C05489=1201.609,-125.840,-37.789,179.030,5.510,149.258
C05490=1201.614,-126.089,-37.779,179.027,5.510,149.259
C05491=1201.619,-126.339,-37.770,179.026,5.510,149.259
C05492=1201.624,-126.589,-37.761,179.024,5.510,149.260
C05493=1201.631,-126.838,-37.752,179.022,5.509,149.261
C05494=1201.208,-126.849,-37.790,179.017,5.513,149.263
C05495=1201.203,-126.600,-37.800,179.020,5.513,149.262
C05496=1201.198,-126.350,-37.809,179.021,5.513,149.262
C05497=1201.192,-126.100,-37.818,179.024,5.514,149.261
C05498=1201.187,-125.850,-37.827,179.026,5.513,149.260
C05499=1201.182,-125.601,-37.836,179.028,5.513,149.260
C05500=1201.176,-125.350,-37.845,179.030,5.514,149.259
C05501=1201.171,-125.101,-37.855,179.032,5.514,149.258
C05502=1201.166,-124.851,-37.864,179.035,5.514,149.258
C05503=1201.161,-124.601,-37.873,179.037,5.514,149.257
C05504=1201.155,-124.351,-37.882,179.039,5.515,149.257
C05505=1201.150,-124.101,-37.891,179.041,5.514,149.256
C05506=1201.145,-123.852,-37.901,179.044,5.515,149.255
C05507=1201.140,-123.602,-37.910,179.045,5.515,149.255
C05508=1201.134,-123.352,-37.919,179.048,5.515,149.254
C05509=1201.129,-123.102,-37.928,179.050,5.515,149.253
C05510=1201.124,-122.853,-37.938,179.052,5.515,149.253
C05511=1201.118,-122.603,-37.947,179.054,5.515,149.252
C05512=1201.113,-122.353,-37.956,179.057,5.516,149.251
C05513=1201.108,-122.103,-37.965,179.059,5.515,149.251
C05514=1201.103,-121.854,-37.974,179.060,5.515,149.250
C05515=1201.097,-121.604,-37.984,179.063,5.516,149.250
C05516=1201.092,-121.354,-37.993,179.065,5.515,149.249
C05517=1201.087,-121.105,-38.002,179.067,5.516,149.248
C05518=1201.081,-120.855,-38.012,179.069,5.516,149.248
C05519=1201.076,-120.605,-38.021,179.072,5.516,149.247
C05520=1201.071,-120.355,-38.030,179.074,5.516,149.246
C05521=1201.065,-120.105,-38.040,179.076,5.516,149.246
C05522=1201.060,-119.855,-38.049,179.078,5.516,149.245
C05523=1201.055,-119.606,-38.058,179.081,5.517,149.245
C05524=1201.049,-119.356,-38.068,179.083,5.516,149.244
C05525=1201.044,-119.106,-38.077,179.085,5.517,149.243
C05526=1201.039,-118.857,-38.086,179.087,5.517,149.243
C05527=1201.033,-118.607,-38.096,179.090,5.517,149.242
C05528=1201.028,-118.357,-38.105,179.091,5.517,149.241
C05529=1201.023,-118.108,-38.114,179.094,5.518,149.241
C05530=1201.017,-117.858,-38.124,179.096,5.517,149.240
C05531=1201.012,-117.608,-38.134,179.098,5.518,149.239
C05532=1201.007,-117.358,-38.143,179.100,5.518,149.239
C05533=1201.001,-117.108,-38.152,179.102,5.518,149.238
C05534=1200.997,-116.859,-38.162,179.105,5.518,149.238
C05535=1200.991,-116.608,-38.171,179.107,5.518,149.237
C05536=1200.986,-116.359,-38.181,179.109,5.518,149.236
C05537=1200.980,-116.109,-38.191,179.111,5.518,149.236
C05538=1200.975,-115.859,-38.199,179.114,5.518,149.235
C05539=1200.970,-115.610,-38.209,179.115,5.518,149.234
C05540=1200.965,-115.360,-38.219,179.118,5.519,149.234
C05541=1200.960,-115.110,-38.228,179.120,5.518,149.233
C05542=1200.954,-114.860,-38.238,179.122,5.519,149.233
C05543=1200.949,-114.611,-38.247,179.124,5.519,149.232
C05544=1200.943,-114.361,-38.257,179.127,5.519,149.231
C05545=1200.938,-114.112,-38.266,179.128,5.519,149.231
C05546=1200.932,-113.861,-38.276,179.131,5.520,149.230
C05547=1200.928,-113.611,-38.286,179.133,5.519,149.229
C05548=1200.923,-113.362,-38.295,179.135,5.520,149.229
C05549=1200.917,-113.112,-38.305,179.138,5.520,149.228
C05550=1200.912,-112.862,-38.314,179.140,5.520,149.227
C05551=1200.906,-112.613,-38.324,179.142,5.520,149.227
C05552=1200.901,-112.363,-38.333,179.145,5.520,149.226
C05553=1200.896,-112.113,-38.343,179.147,5.520,149.225
C05554=1200.890,-111.863,-38.352,179.149,5.521,149.225
C05555=1200.885,-111.614,-38.362,179.151,5.520,149.224
C05556=1200.880,-111.363,-38.372,179.153,5.521,149.224
C05557=1200.875,-111.114,-38.382,179.155,5.521,149.223
C05558=1200.870,-110.865,-38.391,179.158,5.521,149.222
C05559=1200.864,-110.614,-38.401,179.160,5.521,149.222
C05560=1200.859,-110.365,-38.410,179.162,5.522,149.221
C05561=1200.853,-110.115,-38.420,179.164,5.521,149.220
C05562=1200.848,-109.866,-38.430,179.167,5.522,149.220
C05563=1200.843,-109.615,-38.439,179.168,5.522,149.219
C05564=1200.838,-109.366,-38.449,179.171,5.522,149.218
C05565=1200.833,-109.116,-38.459,179.173,5.522,149.218
C05566=1200.827,-108.866,-38.469,179.175,5.522,149.217
C05567=1200.822,-108.617,-38.478,179.178,5.522,149.217
C05568=1200.816,-108.367,-38.489,179.180,5.522,149.216
C05569=1200.812,-108.117,-38.498,179.182,5.522,149.215
C05570=1200.806,-107.867,-38.508,179.184,5.523,149.215
C05571=1200.801,-107.618,-38.518,179.187,5.522,149.214
C05572=1200.795,-107.368,-38.527,179.189,5.523,149.213
C05573=1200.790,-107.118,-38.537,179.191,5.523,149.213
C05574=1200.785,-106.868,-38.547,179.194,5.523,149.212
C05575=1200.780,-106.618,-38.557,179.195,5.523,149.211
C05576=1200.775,-106.369,-38.566,179.198,5.524,149.211
C05577=1200.769,-106.119,-38.577,179.200,5.523,149.210
C05578=1200.764,-105.869,-38.586,179.202,5.524,149.210
C05579=1200.759,-105.619,-38.596,179.204,5.524,149.209
C05580=1200.753,-105.370,-38.606,179.207,5.524,149.208
C05581=1200.748,-105.120,-38.615,179.208,5.524,149.208
C05582=1200.743,-104.870,-38.625,179.211,5.524,149.207
C05583=1200.737,-104.621,-38.636,179.213,5.524,149.206
C05584=1200.733,-104.371,-38.646,179.216,5.525,149.206
C05585=1200.727,-104.121,-38.655,179.217,5.525,149.205
C05586=1200.722,-103.871,-38.665,179.220,5.525,149.204
C05587=1200.716,-103.622,-38.675,179.222,5.525,149.204
C05588=1200.711,-103.372,-38.685,179.224,5.525,149.203
C05589=1200.706,-103.122,-38.694,179.226,5.525,149.202
C05590=1200.701,-102.872,-38.705,179.229,5.525,149.202
C05591=1200.695,-102.623,-38.715,179.231,5.525,149.201
C05592=1200.691,-102.373,-38.725,179.233,5.526,149.200
C05593=1200.685,-102.123,-38.735,179.236,5.525,149.200
C05594=1200.679,-101.873,-38.744,179.238,5.526,149.199
C05595=1200.674,-101.602,-38.755,179.240,5.527,149.199
C05596=1200.669,-101.330,-38.766,179.242,5.526,149.198
C05597=1200.662,-101.060,-38.778,179.245,5.527,149.197
C05598=1200.657,-100.788,-38.788,179.248,5.527,149.196
C05599=1200.651,-100.538,-38.798,179.250,5.527,149.196
C05600=1200.646,-100.288,-38.809,179.253,5.527,149.195
C05601=1200.641,-100.039,-38.818,179.254,5.527,149.195
C05602=1200.636,-99.789,-38.828,179.257,5.527,149.194
C05603=1200.631,-99.539,-38.839,179.259,5.527,149.193
C05604=1200.626,-99.289,-38.848,179.262,5.527,149.192
C05605=1200.620,-99.039,-38.858,179.263,5.527,149.192
C05606=1200.614,-98.790,-38.868,179.266,5.528,149.191
C05607=1200.609,-98.540,-38.879,179.268,5.527,149.190
C05608=1200.605,-98.290,-38.888,179.270,5.528,149.190
C05609=1200.599,-98.041,-38.899,179.272,5.528,149.189
C05610=1200.594,-97.791,-38.909,179.275,5.528,149.189
C05611=1200.588,-97.541,-38.919,179.277,5.528,149.188
C05612=1200.583,-97.292,-38.930,179.279,5.529,149.187
C05613=1200.578,-97.042,-38.940,179.282,5.529,149.187
C05614=1200.573,-96.792,-38.950,179.284,5.529,149.186
C05615=1200.567,-96.542,-38.959,179.286,5.530,149.185
C05616=1200.562,-96.292,-38.970,179.288,5.529,149.185
C05617=1200.556,-96.042,-38.980,179.291,5.530,149.184
C05618=1200.552,-95.793,-38.990,179.293,5.529,149.183
C05619=1200.547,-95.543,-39.000,179.295,5.530,149.183
C05620=1200.541,-95.293,-39.011,179.297,5.530,149.182
C05621=1200.535,-95.044,-39.021,179.300,5.530,149.181
C05622=1200.530,-94.793,-39.031,179.302,5.530,149.181
C05623=1200.525,-94.544,-39.041,179.304,5.530,149.180
C05624=1200.520,-94.295,-39.051,179.306,5.530,149.180
C05625=1200.515,-94.044,-39.062,179.309,5.530,149.179
C05626=1200.509,-93.795,-39.072,179.311,5.530,149.178
C05627=1200.504,-93.545,-39.082,179.313,5.531,149.178
C05628=1200.499,-93.295,-39.093,179.316,5.531,149.177
C05629=1200.494,-93.046,-39.102,179.318,5.531,149.176
C05630=1200.489,-92.796,-39.114,179.320,5.532,149.176
C05631=1200.484,-92.547,-39.124,179.322,5.531,149.175
C05632=1200.478,-92.297,-39.134,179.325,5.532,149.174
C05633=1200.473,-92.047,-39.145,179.327,5.532,149.174
C05634=1200.467,-91.797,-39.155,179.329,5.532,149.173
C05635=1200.462,-91.548,-39.165,179.331,5.532,149.172
C05636=1200.457,-91.297,-39.176,179.334,5.532,149.172
C05637=1200.452,-91.048,-39.185,179.336,5.532,149.171
C05638=1200.447,-90.798,-39.196,179.338,5.533,149.170
C05639=1200.441,-90.548,-39.206,179.341,5.533,149.170
C05640=1200.436,-90.299,-39.216,179.343,5.533,149.169
C05641=1200.431,-90.049,-39.227,179.345,5.533,149.169
C05642=1200.425,-89.800,-39.238,179.347,5.533,149.168
C05643=1200.420,-89.549,-39.248,179.350,5.534,149.167
C05644=1200.415,-89.300,-39.258,179.352,5.533,149.166
C05645=1200.410,-89.050,-39.269,179.354,5.534,149.166
C05646=1200.404,-88.800,-39.279,179.356,5.534,149.165
C05647=1200.399,-88.551,-39.289,179.359,5.534,149.165
C05648=1200.394,-88.301,-39.301,179.361,5.534,149.164
C05649=1200.388,-88.051,-39.311,179.363,5.534,149.163
C05650=1200.383,-87.801,-39.322,179.366,5.535,149.163
C05651=1200.378,-87.552,-39.331,179.368,5.534,149.162
C05652=1200.373,-87.302,-39.342,179.371,5.535,149.161
C05653=1200.368,-87.053,-39.353,179.372,5.535,149.161
C05654=1200.363,-86.803,-39.363,179.375,5.535,149.160
C05655=1200.358,-86.553,-39.373,179.377,5.535,149.159
C05656=1200.353,-86.303,-39.384,179.380,5.535,149.159
C05657=1200.347,-86.054,-39.395,179.382,5.536,149.158
C05658=1200.342,-85.804,-39.405,179.384,5.536,149.157
C05659=1200.337,-85.554,-39.416,179.387,5.536,149.157
C05660=1200.331,-85.304,-39.426,179.389,5.536,149.156
C05661=1200.326,-85.055,-39.437,179.391,5.537,149.156
C05662=1200.321,-84.805,-39.447,179.393,5.536,149.155
C05663=1200.316,-84.555,-39.458,179.396,5.537,149.154
C05664=1200.310,-84.306,-39.468,179.398,5.536,149.153
C05665=1200.305,-84.056,-39.479,179.400,5.537,149.153
C05666=1200.300,-83.806,-39.490,179.403,5.538,149.152
C05667=1200.295,-83.556,-39.500,179.405,5.537,149.151
C05668=1200.290,-83.307,-39.511,179.407,5.538,149.151
C05669=1200.284,-83.057,-39.522,179.409,5.538,149.150
C05670=1200.278,-82.807,-39.533,179.412,5.538,149.150
C05671=1200.274,-82.557,-39.544,179.414,5.538,149.149
C05672=1200.269,-82.307,-39.554,179.416,5.538,149.148
C05673=1200.263,-82.058,-39.565,179.419,5.539,149.148
C05674=1200.258,-81.808,-39.576,179.421,5.538,149.147
C05675=1200.253,-81.558,-39.586,179.423,5.539,149.146
C05676=1200.248,-81.308,-39.597,179.425,5.539,149.146
C05677=1200.242,-81.059,-39.608,179.428,5.539,149.145
C05678=1200.237,-80.809,-39.618,179.430,5.539,149.144
C05679=1200.232,-80.560,-39.629,179.432,5.539,149.144
C05680=1200.227,-80.310,-39.640,179.435,5.540,149.143
C05681=1200.221,-80.060,-39.651,179.437,5.539,149.142
C05682=1200.216,-79.810,-39.662,179.439,5.540,149.142
C05683=1200.210,-79.561,-39.672,179.441,5.540,149.141
C05684=1200.206,-79.311,-39.683,179.444,5.540,149.140
C05685=1200.201,-79.061,-39.694,179.447,5.541,149.140
C05686=1200.195,-78.811,-39.704,179.448,5.541,149.139
C05687=1200.191,-78.562,-39.715,179.451,5.541,149.138
C05688=1200.185,-78.312,-39.726,179.453,5.541,149.138
C05689=1200.179,-78.062,-39.737,179.456,5.541,149.137
C05690=1200.174,-77.813,-39.748,179.457,5.541,149.137
C05691=1200.169,-77.563,-39.759,179.460,5.542,149.136
C05692=1200.164,-77.313,-39.770,179.463,5.542,149.135
C05693=1200.159,-77.064,-39.780,179.465,5.542,149.134
C05694=1200.154,-76.814,-39.791,179.468,5.542,149.134
C05695=1200.148,-76.565,-39.803,179.469,5.542,149.133
C05696=1200.143,-76.314,-39.813,179.472,5.543,149.133
C05697=1200.138,-76.065,-39.824,179.474,5.543,149.132
C05698=1200.133,-75.815,-39.835,179.477,5.543,149.131
C05699=1200.127,-75.544,-39.847,179.479,5.543,149.130
C05700=1200.121,-75.274,-39.859,179.482,5.544,149.130
C05701=1200.116,-75.003,-39.870,179.484,5.543,149.129
C05702=1200.110,-74.732,-39.883,179.487,5.544,149.128
C05703=1200.105,-74.483,-39.893,179.489,5.544,149.128
C05704=1200.099,-74.233,-39.905,179.491,5.544,149.127
C05705=1200.094,-73.982,-39.915,179.494,5.544,149.126
C05706=1200.089,-73.734,-39.926,179.496,5.544,149.126
C05707=1200.084,-73.484,-39.938,179.498,5.545,149.125
C05708=1200.078,-73.234,-39.948,179.501,5.545,149.124
C05709=1200.073,-72.984,-39.960,179.503,5.545,149.124
C05710=1200.068,-72.734,-39.970,179.505,5.545,149.123
C05711=1200.063,-72.485,-39.981,179.507,5.545,149.122
C05712=1200.058,-72.235,-39.993,179.510,5.545,149.122
C05713=1200.053,-71.985,-40.004,179.512,5.546,149.121
C05714=1200.047,-71.736,-40.015,179.514,5.546,149.120
C05715=1200.041,-71.486,-40.026,179.517,5.546,149.120
C05716=1200.037,-71.236,-40.037,179.519,5.546,149.119
C05717=1200.031,-70.987,-40.048,179.521,5.547,149.119
C05718=1200.026,-70.737,-40.058,179.524,5.547,149.118
C05719=1200.021,-70.487,-40.070,179.526,5.547,149.117
C05720=1200.016,-70.238,-40.081,179.529,5.547,149.116
C05721=1200.011,-69.988,-40.092,179.531,5.548,149.116
C05722=1200.005,-69.738,-40.104,179.533,5.548,149.115
C05723=1200.000,-69.489,-40.115,179.536,5.548,149.115
C05724=1199.995,-69.239,-40.126,179.538,5.548,149.114
C05725=1199.990,-68.989,-40.137,179.540,5.548,149.113
C05726=1199.984,-68.740,-40.148,179.543,5.549,149.112
C05727=1199.980,-68.490,-40.159,179.545,5.549,149.112
C05728=1199.974,-68.240,-40.171,179.547,5.549,149.111
C05729=1199.969,-67.990,-40.182,179.549,5.549,149.111
C05730=1199.963,-67.741,-40.193,179.552,5.549,149.110
C05731=1199.958,-67.491,-40.205,179.555,5.550,149.109
C05732=1199.953,-67.241,-40.215,179.556,5.550,149.109
C05733=1199.947,-66.992,-40.227,179.559,5.550,149.108
C05734=1199.943,-66.742,-40.238,179.562,5.551,149.107
C05735=1199.938,-66.492,-40.249,179.564,5.550,149.107
C05736=1199.933,-66.242,-40.261,179.566,5.551,149.106
C05737=1199.927,-65.993,-40.271,179.568,5.551,149.105
C05738=1199.922,-65.743,-40.283,179.571,5.551,149.105
C05739=1199.917,-65.493,-40.295,179.573,5.551,149.104
C05740=1199.912,-65.244,-40.306,179.575,5.551,149.103
C05741=1199.906,-64.994,-40.317,179.578,5.552,149.103
C05742=1199.902,-64.745,-40.329,179.580,5.552,149.102
C05743=1199.896,-64.494,-40.340,179.582,5.552,149.101
C05744=1199.891,-64.245,-40.351,179.585,5.552,149.101
C05745=1199.885,-63.995,-40.363,179.587,5.552,149.100
C05746=1199.880,-63.746,-40.374,179.590,5.553,149.099
C05747=1199.876,-63.496,-40.385,179.592,5.553,149.099
C05748=1199.870,-63.246,-40.397,179.594,5.553,149.098
C05749=1199.866,-62.997,-40.408,179.597,5.553,149.097
C05750=1199.859,-62.747,-40.419,179.599,5.554,149.097
C05751=1199.855,-62.497,-40.430,179.601,5.553,149.096
C05752=1199.849,-62.247,-40.442,179.604,5.554,149.095
C05753=1199.844,-61.998,-40.454,179.606,5.554,149.095
C05754=1199.838,-61.748,-40.465,179.608,5.554,149.094
C05755=1199.834,-61.499,-40.476,179.611,5.555,149.093
C05756=1199.828,-61.249,-40.488,179.613,5.554,149.093
C05757=1199.824,-60.999,-40.500,179.615,5.555,149.092
C05758=1199.818,-60.749,-40.512,179.618,5.556,149.091
C05759=1199.813,-60.500,-40.523,179.620,5.555,149.091
C05760=1199.807,-60.250,-40.534,179.623,5.556,149.090
C05761=1199.803,-60.001,-40.546,179.625,5.556,149.089
C05762=1199.797,-59.751,-40.558,179.627,5.556,149.089
C05763=1199.793,-59.501,-40.569,179.630,5.557,149.088
C05764=1199.787,-59.251,-40.581,179.632,5.557,149.087
C05765=1199.782,-59.002,-40.592,179.634,5.557,149.087
C05766=1199.776,-58.752,-40.604,179.637,5.557,149.086
C05767=1199.772,-58.503,-40.615,179.639,5.557,149.086
C05768=1199.766,-58.253,-40.627,179.641,5.558,149.085
C05769=1199.761,-58.003,-40.639,179.644,5.558,149.084
C05770=1199.756,-57.753,-40.650,179.646,5.558,149.083
C05771=1199.751,-57.503,-40.662,179.649,5.558,149.083
C05772=1199.746,-57.254,-40.673,179.651,5.559,149.082
C05773=1199.740,-57.004,-40.685,179.653,5.559,149.082
C05774=1199.735,-56.755,-40.696,179.656,5.559,149.081
C05775=1199.730,-56.505,-40.708,179.658,5.560,149.080
C05776=1199.725,-56.255,-40.720,179.660,5.559,149.079
C05777=1199.720,-56.005,-40.731,179.663,5.560,149.079
C05778=1199.714,-55.755,-40.743,179.665,5.561,149.078
C05779=1199.710,-55.506,-40.755,179.667,5.560,149.078
C05780=1199.705,-55.256,-40.767,179.670,5.561,149.077
C05781=1199.699,-55.007,-40.778,179.673,5.561,149.076
C05782=1199.694,-54.758,-40.789,179.675,5.561,149.075
C05783=1199.688,-54.508,-40.801,179.677,5.562,149.075
C05784=1199.684,-54.258,-40.813,179.680,5.562,149.074
C05785=1199.678,-54.008,-40.825,179.682,5.562,149.074
C05786=1199.673,-53.758,-40.836,179.684,5.562,149.073
C05787=1199.668,-53.509,-40.848,179.687,5.562,149.072
C05788=1199.663,-53.259,-40.860,179.689,5.562,149.071
C05789=1199.658,-53.009,-40.872,179.691,5.563,149.071
C05790=1199.653,-52.760,-40.884,179.694,5.563,149.070
C05791=1199.647,-52.510,-40.895,179.696,5.563,149.070
C05792=1199.642,-52.260,-40.908,179.699,5.563,149.069
C05793=1199.638,-52.011,-40.919,179.701,5.564,149.068
C05794=1199.632,-51.762,-40.931,179.703,5.564,149.068
C05795=1199.626,-51.512,-40.943,179.706,5.564,149.067
C05796=1199.622,-51.262,-40.954,179.708,5.565,149.066
C05797=1199.616,-51.013,-40.967,179.710,5.565,149.066
C05798=1199.611,-50.763,-40.978,179.713,5.565,149.065
C05799=1199.606,-50.513,-40.990,179.716,5.565,149.064
C05800=1199.601,-50.263,-41.002,179.717,5.565,149.064
C05801=1199.596,-50.014,-41.014,179.720,5.566,149.063
C05802=1199.590,-49.764,-41.026,179.723,5.566,149.062
C05803=1199.585,-49.494,-41.039,179.725,5.567,149.062
C05804=1199.579,-49.224,-41.052,179.727,5.566,149.061
C05805=1199.574,-48.954,-41.065,179.730,5.567,149.060
C05806=1199.568,-48.683,-41.078,179.733,5.567,149.059
C05807=1199.563,-48.433,-41.090,179.735,5.568,149.059
C05808=1199.558,-48.184,-41.102,179.737,5.567,149.058
C05809=1199.553,-47.934,-41.113,179.740,5.568,149.057
C05810=1199.548,-47.684,-41.125,179.743,5.568,149.057
C05811=1199.543,-47.435,-41.138,179.744,5.568,149.056
C05812=1199.537,-47.185,-41.150,179.747,5.569,149.055
C05813=1199.532,-46.935,-41.162,179.750,5.569,149.055
C05814=1199.527,-46.686,-41.174,179.752,5.569,149.054
C05815=1199.522,-46.436,-41.186,179.754,5.569,149.053
C05816=1199.517,-46.186,-41.197,179.757,5.570,149.053
C05817=1199.511,-45.937,-41.210,179.759,5.571,149.052
C05818=1199.506,-45.687,-41.222,179.761,5.570,149.051
C05819=1199.502,-45.438,-41.234,179.764,5.571,149.051
C05820=1199.496,-45.188,-41.246,179.767,5.571,149.050
C05821=1199.491,-44.938,-41.258,179.769,5.571,149.049
C05822=1199.486,-44.689,-41.270,179.771,5.572,149.049
C05823=1199.480,-44.439,-41.282,179.774,5.572,149.048
C05824=1199.475,-44.190,-41.295,179.776,5.572,149.048
C05825=1199.470,-43.940,-41.307,179.778,5.572,149.047
C05826=1199.465,-43.691,-41.319,179.781,5.573,149.046
C05827=1199.460,-43.441,-41.331,179.784,5.573,149.045
C05828=1199.454,-43.191,-41.342,179.785,5.573,149.045
C05829=1199.449,-42.941,-41.355,179.788,5.574,149.044
C05830=1199.444,-42.692,-41.367,179.791,5.574,149.044
C05831=1199.439,-42.442,-41.380,179.793,5.574,149.043
C05832=1199.433,-42.192,-41.391,179.795,5.574,149.042
C05833=1199.428,-41.943,-41.404,179.798,5.575,149.042
C05834=1199.423,-41.693,-41.415,179.800,5.575,149.041
C05835=1199.419,-41.443,-41.428,179.802,5.575,149.040
C05836=1199.414,-41.193,-41.440,179.805,5.576,149.040
C05837=1199.408,-40.944,-41.453,179.808,5.576,149.039
C05838=1199.403,-40.695,-41.465,179.810,5.576,149.038
C05839=1199.398,-40.445,-41.477,179.812,5.577,149.038
C05840=1199.393,-40.195,-41.490,179.815,5.577,149.037
C05841=1199.387,-39.946,-41.502,179.817,5.577,149.036
C05842=1199.382,-39.696,-41.514,179.819,5.577,149.036
C05843=1199.377,-39.446,-41.526,179.822,5.578,149.035
C05844=1199.372,-39.197,-41.539,179.825,5.578,149.034
C05845=1199.367,-38.947,-41.552,179.826,5.578,149.034
C05846=1199.362,-38.697,-41.564,179.829,5.579,149.033
C05847=1199.357,-38.448,-41.576,179.832,5.579,149.032
C05848=1199.351,-38.198,-41.588,179.834,5.579,149.032
C05849=1199.346,-37.948,-41.601,179.836,5.579,149.031
C05850=1199.341,-37.699,-41.613,179.839,5.580,149.030
C05851=1199.335,-37.449,-41.625,179.841,5.580,149.030
C05852=1199.330,-37.200,-41.638,179.843,5.580,149.029
C05853=1199.325,-36.949,-41.650,179.846,5.581,149.028
C05854=1199.320,-36.700,-41.663,179.849,5.581,149.028
C05855=1199.315,-36.451,-41.675,179.851,5.581,149.027
C05856=1199.310,-36.201,-41.687,179.853,5.581,149.026
C05857=1199.305,-35.951,-41.700,179.855,5.582,149.026
C05858=1199.300,-35.702,-41.712,179.858,5.582,149.025
C05859=1199.295,-35.452,-41.725,179.861,5.583,149.024
C05860=1199.290,-35.202,-41.737,179.863,5.582,149.024
C05861=1199.284,-34.953,-41.750,179.866,5.583,149.023
C05862=1199.279,-34.703,-41.762,179.868,5.583,149.022
C05863=1199.274,-34.453,-41.774,179.870,5.583,149.022
C05864=1199.269,-34.204,-41.787,179.872,5.584,149.021
C05865=1199.264,-33.954,-41.800,179.875,5.584,149.020
C05866=1199.259,-33.705,-41.812,179.878,5.585,149.020
C05867=1199.254,-33.455,-41.824,179.880,5.584,149.019
C05868=1199.248,-33.205,-41.838,179.883,5.585,149.018
C05869=1199.243,-32.956,-41.850,179.885,5.586,149.018
C05870=1199.238,-32.706,-41.863,179.887,5.586,149.017
C05871=1199.233,-32.456,-41.875,179.889,5.586,149.016
C05872=1199.228,-32.207,-41.888,179.892,5.586,149.016
C05873=1199.223,-31.957,-41.900,179.895,5.587,149.015
C05874=1199.217,-31.708,-41.913,179.897,5.587,149.014
C05875=1199.213,-31.458,-41.926,179.899,5.587,149.014
C05876=1199.208,-31.209,-41.938,179.902,5.588,149.013
C05877=1199.202,-30.958,-41.951,179.904,5.588,149.012
C05878=1199.196,-30.709,-41.963,179.907,5.589,149.012
C05879=1199.192,-30.459,-41.976,179.909,5.588,149.011
C05880=1199.187,-30.210,-41.989,179.911,5.589,149.011
C05881=1199.182,-29.960,-42.002,179.914,5.590,149.010
C05882=1199.177,-29.711,-42.014,179.917,5.590,149.009
C05883=1199.172,-29.461,-42.026,179.919,5.590,149.009
C05884=1199.166,-29.211,-42.040,179.921,5.590,149.008
C05885=1199.161,-28.962,-42.052,179.924,5.591,149.007
C05886=1199.156,-28.712,-42.065,179.926,5.592,149.007
C05887=1199.151,-28.462,-42.078,179.928,5.591,149.006
C05888=1199.146,-28.213,-42.090,179.931,5.592,149.005
C05889=1199.140,-27.963,-42.104,179.934,5.592,149.005
C05890=1199.136,-27.713,-42.117,179.936,5.593,149.004
C05891=1199.131,-27.464,-42.129,179.939,5.593,149.003
C05892=1199.125,-27.215,-42.142,179.940,5.593,149.003
C05893=1199.120,-26.965,-42.154,179.943,5.594,149.002
C05894=1199.115,-26.715,-42.168,179.946,5.594,149.001
C05895=1199.110,-26.466,-42.181,179.948,5.595,149.001
C05896=1199.105,-26.216,-42.193,179.950,5.594,149.000
C05897=1199.100,-25.966,-42.206,179.953,5.595,148.999
C05898=1199.094,-25.717,-42.219,179.955,5.596,148.999
C05899=1199.089,-25.467,-42.232,179.958,5.596,148.998
C05900=1199.085,-25.217,-42.245,179.960,5.596,148.997
C05901=1199.080,-24.968,-42.258,179.963,5.596,148.997
C05902=1199.074,-24.718,-42.271,179.965,5.597,148.996
C05903=1199.069,-24.468,-42.284,179.968,5.597,148.995
C05904=1199.064,-24.219,-42.296,179.970,5.598,148.995
C05905=1199.059,-23.970,-42.309,179.972,5.598,148.994
C05906=1199.054,-23.719,-42.322,179.975,5.598,148.993
C05907=1199.048,-23.450,-42.336,179.978,5.599,148.993
C05908=1199.042,-23.180,-42.350,179.980,5.599,148.992
C05909=1199.037,-22.911,-42.364,179.983,5.600,148.991
C05910=1199.031,-22.641,-42.378,179.986,5.600,148.991
C05911=1199.027,-22.392,-42.391,179.988,5.600,148.990
C05912=1199.022,-22.143,-42.404,179.990,5.600,148.989
C05913=1199.016,-21.893,-42.417,179.993,5.601,148.989
C05914=1199.011,-21.643,-42.430,179.996,5.601,148.988
C05915=1199.005,-21.393,-42.443,179.998,5.602,148.987
C05916=1199.000,-21.144,-42.456,-180.000,5.602,148.987
C05917=1198.996,-20.894,-42.469,-179.997,5.602,148.986
C05918=1198.990,-20.644,-42.482,-179.995,5.603,148.985
C05919=1198.986,-20.395,-42.496,-179.992,5.603,148.985
C05920=1198.981,-20.146,-42.508,-179.989,5.603,148.984
C05921=1198.975,-19.896,-42.521,-179.987,5.604,148.983
C05922=1198.970,-19.646,-42.534,-179.985,5.604,148.983
C05923=1198.964,-19.396,-42.548,-179.983,5.604,148.982
C05924=1198.960,-19.146,-42.561,-179.980,5.605,148.981
C05925=1198.955,-18.898,-42.574,-179.977,5.605,148.981
C05926=1198.949,-18.648,-42.587,-179.975,5.606,148.980
C05927=1198.945,-18.398,-42.600,-179.973,5.606,148.979
C05928=1198.939,-18.148,-42.613,-179.970,5.606,148.979
C05929=1198.935,-17.899,-42.627,-179.968,5.607,148.978
C05930=1198.929,-17.650,-42.640,-179.965,5.607,148.977
C05931=1198.924,-17.400,-42.653,-179.962,5.608,148.977
C05932=1198.919,-17.150,-42.666,-179.960,5.607,148.976
C05933=1198.913,-16.901,-42.680,-179.958,5.608,148.976
C05934=1198.909,-16.651,-42.693,-179.955,5.609,148.975
C05935=1198.903,-16.401,-42.706,-179.953,5.609,148.974
C05936=1198.899,-16.151,-42.719,-179.950,5.610,148.973
C05937=1198.893,-15.902,-42.733,-179.948,5.609,148.973
C05938=1198.888,-15.652,-42.746,-179.945,5.610,148.972
C05939=1198.883,-15.403,-42.758,-179.943,5.611,148.972
C05940=1198.878,-15.153,-42.773,-179.941,5.611,148.971
C05941=1198.873,-14.904,-42.785,-179.938,5.612,148.970
C05942=1198.867,-14.654,-42.798,-179.936,5.611,148.970
C05943=1198.863,-14.405,-42.812,-179.933,5.612,148.969
C05944=1198.857,-14.155,-42.825,-179.931,5.612,148.968
C05945=1198.853,-13.905,-42.838,-179.928,5.613,148.968
C05946=1198.847,-13.656,-42.852,-179.926,5.614,148.967
C05947=1198.842,-13.406,-42.866,-179.923,5.614,148.966
C05948=1198.837,-13.157,-42.878,-179.921,5.614,148.966
C05949=1198.832,-12.907,-42.893,-179.918,5.614,148.965
C05950=1198.827,-12.658,-42.905,-179.916,5.615,148.964
C05951=1198.822,-12.408,-42.919,-179.913,5.616,148.964
C05952=1198.817,-12.159,-42.932,-179.911,5.616,148.963
C05953=1198.812,-11.909,-42.946,-179.908,5.617,148.962
C05954=1198.807,-11.660,-42.959,-179.906,5.616,148.962
C05955=1198.801,-11.409,-42.972,-179.903,5.617,148.961
C05956=1198.797,-11.161,-42.986,-179.901,5.617,148.960
C05957=1198.791,-10.910,-42.999,-179.899,5.618,148.960
C05958=1198.786,-10.660,-43.014,-179.896,5.619,148.959
C05959=1198.781,-10.411,-43.026,-179.893,5.619,148.958
C05960=1198.776,-10.161,-43.040,-179.891,5.619,148.958
C05961=1198.771,-9.912,-43.053,-179.889,5.619,148.957
C05962=1198.766,-9.662,-43.067,-179.886,5.620,148.957
C05963=1198.760,-9.413,-43.081,-179.884,5.621,148.956
C05964=1198.756,-9.163,-43.094,-179.881,5.621,148.955
C05965=1198.750,-8.914,-43.107,-179.878,5.622,148.955
C05966=1198.746,-8.664,-43.121,-179.876,5.621,148.954
C05967=1198.740,-8.415,-43.134,-179.874,5.622,148.953
C05968=1198.735,-8.165,-43.149,-179.872,5.623,148.953
C05969=1198.731,-7.915,-43.162,-179.869,5.623,148.952
C05970=1198.725,-7.666,-43.175,-179.866,5.624,148.951
C05971=1198.720,-7.416,-43.189,-179.864,5.624,148.951
C05972=1198.715,-7.167,-43.202,-179.861,5.624,148.950
C05973=1198.710,-6.917,-43.217,-179.859,5.624,148.949
C05974=1198.705,-6.667,-43.230,-179.857,5.625,148.949
C05975=1198.700,-6.418,-43.243,-179.854,5.625,148.948
C05976=1198.695,-6.168,-43.257,-179.851,5.626,148.947
C05977=1198.689,-5.919,-43.271,-179.849,5.626,148.947
C05978=1198.685,-5.670,-43.285,-179.846,5.627,148.946
C05979=1198.680,-5.419,-43.298,-179.844,5.628,148.946
C05980=1198.674,-5.170,-43.312,-179.842,5.627,148.945
C05981=1198.670,-4.921,-43.326,-179.839,5.628,148.944
C05982=1198.664,-4.671,-43.339,-179.837,5.628,148.943
C05983=1198.659,-4.421,-43.353,-179.834,5.629,148.943
C05984=1198.654,-4.172,-43.368,-179.831,5.629,148.942
C05985=1198.649,-3.922,-43.380,-179.829,5.630,148.942
C05986=1198.644,-3.673,-43.394,-179.826,5.631,148.941
C05987=1198.639,-3.423,-43.409,-179.824,5.630,148.940
C05988=1198.633,-3.173,-43.422,-179.822,5.631,148.940
C05989=1198.629,-2.924,-43.436,-179.819,5.631,148.939
C05990=1198.624,-2.675,-43.450,-179.817,5.632,148.938
C05991=1198.618,-2.425,-43.463,-179.814,5.633,148.938
C05992=1198.613,-2.175,-43.477,-179.812,5.633,148.937
C05993=1198.608,-1.926,-43.491,-179.809,5.634,148.936
C05994=1198.604,-1.676,-43.505,-179.806,5.634,148.936
C05995=1198.598,-1.426,-43.518,-179.804,5.634,148.935
C05996=1198.593,-1.177,-43.532,-179.802,5.635,148.935
C05997=1198.588,-0.927,-43.547,-179.799,5.635,148.934
C05998=1198.584,-0.678,-43.560,-179.797,5.636,148.933
C05999=1198.578,-0.428,-43.574,-179.794,5.636,148.932
C06000=1198.573,-0.179,-43.588,-179.791,5.637,148.932
C06001=1198.568,0.071,-43.602,-179.789,5.638,148.931
C06002=1198.563,0.321,-43.616,-179.787,5.638,148.931
C06003=1198.558,0.569,-43.630,-179.784,5.639,148.930
C06004=1198.553,0.820,-43.643,-179.782,5.638,148.929
C06005=1198.548,1.069,-43.658,-179.779,5.639,148.929
C06006=1198.542,1.318,-43.671,-179.777,5.639,148.928
C06007=1198.537,1.568,-43.686,-179.774,5.640,148.927
C06008=1198.532,1.818,-43.700,-179.772,5.641,148.927
C06009=1198.527,2.067,-43.714,-179.769,5.641,148.926
C06010=1198.523,2.316,-43.728,-179.766,5.642,148.925
C06011=1198.516,2.586,-43.743,-179.764,5.642,148.925
C06012=1198.511,2.855,-43.758,-179.761,5.643,148.924
C06013=1198.506,3.125,-43.773,-179.758,5.643,148.923
C06014=1198.500,3.393,-43.789,-179.756,5.644,148.923
C06015=1198.496,3.642,-43.802,-179.753,5.644,148.922
C06016=1198.491,3.892,-43.816,-179.750,5.645,148.921
C06017=1198.486,4.142,-43.831,-179.748,5.645,148.921
C06018=1198.480,4.391,-43.844,-179.746,5.646,148.920
C06019=1198.475,4.641,-43.858,-179.744,5.646,148.919
C06020=1198.470,4.891,-43.873,-179.741,5.646,148.919
C06021=1198.465,5.141,-43.887,-179.738,5.647,148.918
C06022=1198.460,5.390,-43.901,-179.736,5.647,148.918
C06023=1198.454,5.639,-43.915,-179.733,5.648,148.917
C06024=1198.449,5.889,-43.929,-179.731,5.648,148.916
C06025=1198.445,6.139,-43.944,-179.728,5.649,148.915
C06026=1198.440,6.388,-43.958,-179.725,5.649,148.915
C06027=1198.434,6.637,-43.972,-179.723,5.650,148.914
C06028=1198.429,6.887,-43.986,-179.721,5.651,148.914
C06029=1198.424,7.137,-44.000,-179.718,5.651,148.913
C06030=1198.419,7.387,-44.015,-179.716,5.651,148.912
C06031=1198.414,7.636,-44.029,-179.713,5.651,148.912
C06032=1198.409,7.885,-44.043,-179.711,5.652,148.911
C06033=1198.404,8.134,-44.058,-179.708,5.653,148.910
C06034=1198.399,8.384,-44.072,-179.706,5.653,148.910
C06035=1198.394,8.634,-44.086,-179.703,5.654,148.909
C06036=1198.389,8.883,-44.101,-179.701,5.654,148.908
C06037=1198.384,9.133,-44.115,-179.698,5.655,148.908
C06038=1198.379,9.382,-44.129,-179.696,5.656,148.907
C06039=1198.374,9.632,-44.143,-179.693,5.656,148.907
C06040=1198.369,9.882,-44.157,-179.690,5.657,148.906
C06041=1198.364,10.131,-44.172,-179.688,5.657,148.905
C06042=1198.359,10.380,-44.187,-179.686,5.658,148.905
C06043=1198.354,10.630,-44.201,-179.683,5.659,148.904
C06044=1198.349,10.879,-44.215,-179.681,5.658,148.903
C06045=1198.344,11.129,-44.229,-179.678,5.659,148.903
C06046=1198.339,11.379,-44.243,-179.676,5.659,148.902
C06047=1198.334,11.628,-44.258,-179.673,5.660,148.902
C06048=1198.329,11.877,-44.273,-179.671,5.661,148.901
C06049=1198.323,12.127,-44.287,-179.668,5.661,148.900
C06050=1198.318,12.377,-44.302,-179.665,5.662,148.899
C06051=1198.313,12.627,-44.316,-179.663,5.662,148.899
C06052=1198.308,12.876,-44.330,-179.661,5.663,148.898
C06053=1198.303,13.125,-44.345,-179.658,5.663,148.898
C06054=1198.298,13.375,-44.359,-179.655,5.664,148.897
C06055=1198.293,13.624,-44.373,-179.653,5.664,148.896
C06056=1198.288,13.874,-44.388,-179.650,5.665,148.896
C06057=1198.283,14.123,-44.403,-179.648,5.666,148.895
C06058=1198.278,14.373,-44.418,-179.645,5.666,148.894
C06059=1198.273,14.623,-44.432,-179.643,5.667,148.894
C06060=1198.268,14.873,-44.446,-179.640,5.667,148.893
C06061=1198.263,15.122,-44.461,-179.637,5.668,148.892
C06062=1198.258,15.371,-44.475,-179.636,5.668,148.892
C06063=1198.252,15.621,-44.490,-179.633,5.668,148.891
C06064=1198.248,15.870,-44.505,-179.630,5.669,148.891
C06065=1198.243,16.119,-44.519,-179.628,5.669,148.890
C06066=1198.238,16.369,-44.533,-179.626,5.670,148.889
C06067=1198.233,16.618,-44.548,-179.623,5.671,148.889
C06068=1198.227,16.868,-44.563,-179.620,5.671,148.888
C06069=1198.222,17.118,-44.578,-179.618,5.672,148.887
C06070=1198.218,17.367,-44.593,-179.615,5.672,148.887
C06071=1198.213,17.617,-44.607,-179.613,5.673,148.886
C06072=1198.207,17.867,-44.622,-179.610,5.674,148.886
C06073=1198.202,18.116,-44.637,-179.608,5.674,148.885
C06074=1198.197,18.366,-44.651,-179.605,5.675,148.884
C06075=1198.193,18.615,-44.666,-179.602,5.675,148.884
C06076=1198.188,18.864,-44.680,-179.600,5.676,148.883
C06077=1198.182,19.114,-44.695,-179.597,5.677,148.882
C06078=1198.178,19.364,-44.710,-179.595,5.677,148.882
C06079=1198.173,19.613,-44.724,-179.592,5.678,148.881
C06080=1198.167,19.863,-44.740,-179.590,5.678,148.881
C06081=1198.162,20.112,-44.754,-179.587,5.679,148.880
C06082=1198.158,20.361,-44.769,-179.585,5.680,148.879
C06083=1198.153,20.611,-44.784,-179.582,5.680,148.879
C06084=1198.147,20.861,-44.799,-179.579,5.681,148.878
C06085=1198.142,21.110,-44.813,-179.577,5.681,148.877
C06086=1198.138,21.359,-44.828,-179.575,5.682,148.877
C06087=1198.132,21.609,-44.843,-179.572,5.682,148.876
C06088=1198.127,21.858,-44.858,-179.569,5.683,148.875
C06089=1198.122,22.108,-44.873,-179.567,5.683,148.875
C06090=1198.117,22.358,-44.888,-179.565,5.684,148.874
C06091=1198.112,22.607,-44.902,-179.562,5.685,148.874
C06092=1198.107,22.856,-44.917,-179.559,5.685,148.873
C06093=1198.102,23.106,-44.932,-179.557,5.686,148.872
C06094=1198.097,23.356,-44.947,-179.554,5.687,148.872
C06095=1198.092,23.605,-44.962,-179.552,5.687,148.871
C06096=1198.087,23.855,-44.977,-179.549,5.688,148.870
C06097=1198.082,24.104,-44.992,-179.546,5.688,148.870
C06098=1198.076,24.354,-45.007,-179.544,5.689,148.869
C06099=1198.072,24.603,-45.022,-179.542,5.690,148.869
C06100=1198.067,24.852,-45.037,-179.539,5.690,148.868
C06101=1198.061,25.102,-45.052,-179.536,5.691,148.867
C06102=1198.057,25.351,-45.067,-179.534,5.691,148.867
C06103=1198.052,25.602,-45.082,-179.532,5.692,148.866
C06104=1198.047,25.851,-45.097,-179.529,5.693,148.865
C06105=1198.042,26.100,-45.112,-179.526,5.693,148.865
C06106=1198.037,26.350,-45.127,-179.524,5.694,148.864
C06107=1198.032,26.599,-45.142,-179.521,5.694,148.864
C06108=1198.027,26.848,-45.158,-179.519,5.695,148.863
C06109=1198.022,27.098,-45.172,-179.516,5.695,148.862
C06110=1198.016,27.348,-45.187,-179.514,5.696,148.862
C06111=1198.012,27.597,-45.202,-179.511,5.697,148.861
C06112=1198.006,27.846,-45.218,-179.509,5.697,148.860
C06113=1198.002,28.096,-45.233,-179.506,5.698,148.860
C06114=1197.996,28.346,-45.248,-179.503,5.698,148.859
C06115=1197.991,28.615,-45.264,-179.501,5.699,148.858
C06116=1197.986,28.883,-45.281,-179.498,5.699,148.858
C06117=1197.981,29.152,-45.297,-179.496,5.700,148.857
C06118=1197.975,29.420,-45.314,-179.492,5.701,148.856
C06119=1197.970,29.670,-45.328,-179.490,5.702,148.856
C06120=1197.965,29.920,-45.344,-179.487,5.703,148.855
C06121=1197.960,30.169,-45.359,-179.485,5.703,148.855
C06122=1197.955,30.418,-45.374,-179.482,5.704,148.854
C06123=1197.951,30.668,-45.390,-179.480,5.705,148.853
C06124=1197.945,30.918,-45.404,-179.477,5.705,148.853
C06125=1197.940,31.167,-45.420,-179.475,5.706,148.852
C06126=1197.935,31.416,-45.435,-179.472,5.706,148.851
C06127=1197.930,31.666,-45.451,-179.470,5.707,148.851
C06128=1197.925,31.915,-45.466,-179.467,5.708,148.850
C06129=1197.920,32.165,-45.481,-179.465,5.708,148.850
C06130=1197.915,32.414,-45.496,-179.462,5.709,148.849
C06131=1197.910,32.664,-45.511,-179.460,5.709,148.848
C06132=1197.904,32.913,-45.527,-179.457,5.710,148.848
C06133=1197.900,33.163,-45.542,-179.455,5.710,148.847
C06134=1197.895,33.413,-45.558,-179.452,5.711,148.846
C06135=1197.890,33.662,-45.573,-179.450,5.712,148.846
C06136=1197.885,33.911,-45.588,-179.447,5.712,148.845
C06137=1197.880,34.161,-45.604,-179.444,5.713,148.845
C06138=1197.875,34.410,-45.619,-179.442,5.713,148.844
C06139=1197.870,34.660,-45.635,-179.440,5.714,148.844
C06140=1197.865,34.909,-45.650,-179.436,5.716,148.843
C06141=1197.860,35.158,-45.666,-179.434,5.716,148.842
C06142=1197.855,35.408,-45.681,-179.431,5.717,148.842
C06143=1197.851,35.657,-45.697,-179.429,5.718,148.841
C06144=1197.845,35.907,-45.712,-179.426,5.718,148.840
C06145=1197.840,36.156,-45.728,-179.424,5.719,148.840
C06146=1197.835,36.405,-45.743,-179.421,5.719,148.839
C06147=1197.830,36.655,-45.759,-179.419,5.720,148.839
C06148=1197.825,36.905,-45.774,-179.416,5.721,148.838
C06149=1197.820,37.154,-45.790,-179.414,5.721,148.837
C06150=1197.815,37.403,-45.805,-179.411,5.722,148.837
C06151=1197.810,37.653,-45.821,-179.409,5.722,148.836
C06152=1197.805,37.903,-45.836,-179.406,5.723,148.835
C06153=1197.800,38.152,-45.851,-179.404,5.724,148.835
C06154=1197.795,38.401,-45.867,-179.401,5.724,148.834
C06155=1197.790,38.651,-45.883,-179.399,5.725,148.834
C06156=1197.785,38.901,-45.898,-179.396,5.726,148.833
C06157=1197.780,39.150,-45.913,-179.393,5.727,148.832
C06158=1197.775,39.400,-45.929,-179.390,5.727,148.832
C06159=1197.770,39.649,-45.946,-179.388,5.728,148.831
C06160=1197.765,39.898,-45.961,-179.385,5.729,148.831
C06161=1197.760,40.147,-45.976,-179.383,5.729,148.830
C06162=1197.755,40.397,-45.992,-179.381,5.730,148.829
C06163=1197.750,40.647,-46.008,-179.378,5.731,148.829
C06164=1197.745,40.896,-46.023,-179.375,5.731,148.828
C06165=1197.740,41.146,-46.039,-179.373,5.732,148.827
C06166=1197.735,41.395,-46.055,-179.371,5.733,148.827
C06167=1197.730,41.644,-46.071,-179.368,5.733,148.826
C06168=1197.725,41.894,-46.087,-179.365,5.734,148.826
C06169=1197.720,42.144,-46.102,-179.362,5.735,148.825
C06170=1197.714,42.393,-46.118,-179.360,5.736,148.824
C06171=1197.711,42.642,-46.134,-179.357,5.736,148.824
C06172=1197.705,42.892,-46.149,-179.355,5.737,148.823
C06173=1197.700,43.141,-46.165,-179.353,5.738,148.823
C06174=1197.695,43.391,-46.181,-179.350,5.738,148.822
C06175=1197.690,43.640,-46.197,-179.347,5.739,148.821
C06176=1197.685,43.890,-46.213,-179.345,5.739,148.821
C06177=1197.681,44.139,-46.228,-179.342,5.740,148.820
C06178=1197.675,44.389,-46.244,-179.339,5.742,148.820
C06179=1197.671,44.638,-46.261,-179.337,5.742,148.819
C06180=1197.665,44.887,-46.276,-179.334,5.743,148.818
C06181=1197.660,45.137,-46.292,-179.332,5.744,148.818
C06182=1197.655,45.386,-46.308,-179.329,5.744,148.817
C06183=1197.650,45.636,-46.324,-179.327,5.745,148.816
C06184=1197.645,45.886,-46.340,-179.324,5.746,148.816
C06185=1197.640,46.135,-46.356,-179.322,5.746,148.815
C06186=1197.636,46.384,-46.371,-179.319,5.747,148.815
C06187=1197.631,46.634,-46.387,-179.316,5.748,148.814
C06188=1197.626,46.883,-46.403,-179.314,5.749,148.814
C06189=1197.621,47.133,-46.419,-179.311,5.749,148.813
C06190=1197.616,47.381,-46.436,-179.308,5.750,148.812
C06191=1197.611,47.632,-46.452,-179.306,5.751,148.812
C06192=1197.606,47.881,-46.467,-179.304,5.751,148.811
C06193=1197.601,48.130,-46.484,-179.301,5.752,148.810
C06194=1197.596,48.380,-46.500,-179.299,5.753,148.810
C06195=1197.591,48.629,-46.516,-179.296,5.754,148.809
C06196=1197.586,48.879,-46.532,-179.293,5.755,148.809
C06197=1197.581,49.128,-46.548,-179.290,5.755,148.808
C06198=1197.576,49.378,-46.564,-179.288,5.756,148.808
C06199=1197.571,49.627,-46.580,-179.286,5.757,148.807
C06200=1197.566,49.877,-46.596,-179.283,5.757,148.806
C06201=1197.561,50.126,-46.612,-179.281,5.758,148.806
C06202=1197.556,50.375,-46.629,-179.278,5.759,148.805
C06203=1197.551,50.625,-46.644,-179.275,5.760,148.804
C06204=1197.546,50.874,-46.660,-179.273,5.761,148.804
C06205=1197.541,51.124,-46.676,-179.270,5.761,148.803
C06206=1197.536,51.372,-46.693,-179.268,5.762,148.803
C06207=1197.532,51.622,-46.709,-179.265,5.762,148.802
C06208=1197.526,51.871,-46.725,-179.263,5.763,148.802
C06209=1197.522,52.121,-46.742,-179.260,5.764,148.801
C06210=1197.516,52.370,-46.757,-179.257,5.765,148.800
C06211=1197.512,52.620,-46.774,-179.255,5.766,148.800
C06212=1197.506,52.869,-46.789,-179.252,5.767,148.799
C06213=1197.502,53.119,-46.806,-179.249,5.767,148.798
C06214=1197.497,53.368,-46.823,-179.247,5.768,148.798
C06215=1197.491,53.618,-46.839,-179.245,5.769,148.797
C06216=1197.487,53.867,-46.856,-179.242,5.769,148.797
C06217=1197.481,54.117,-46.871,-179.239,5.771,148.796
C06218=1197.477,54.366,-46.888,-179.237,5.771,148.796
C06219=1197.472,54.634,-46.906,-179.234,5.772,148.795
C06220=1197.466,54.903,-46.923,-179.231,5.772,148.794
C06221=1197.461,55.172,-46.940,-179.228,5.774,148.794
C06222=1197.455,55.440,-46.958,-179.226,5.774,148.793
C06223=1197.451,55.689,-46.975,-179.223,5.775,148.792
C06224=1197.445,55.939,-46.991,-179.221,5.776,148.792
C06225=1197.441,56.188,-47.007,-179.218,5.777,148.791
C06226=1197.436,56.437,-47.024,-179.215,5.778,148.791
C06227=1197.431,56.687,-47.040,-179.213,5.778,148.790
C06228=1197.425,56.936,-47.056,-179.210,5.779,148.789
C06229=1197.421,57.186,-47.073,-179.208,5.780,148.789
C06230=1197.416,57.435,-47.090,-179.205,5.780,148.788
C06231=1197.411,57.685,-47.105,-179.202,5.782,148.788
C06232=1197.406,57.934,-47.122,-179.200,5.783,148.787
C06233=1197.401,58.183,-47.139,-179.197,5.783,148.786
C06234=1197.396,58.433,-47.156,-179.195,5.784,148.786
C06235=1197.391,58.683,-47.172,-179.193,5.785,148.785
C06236=1197.386,58.932,-47.188,-179.189,5.786,148.785
C06237=1197.382,59.181,-47.205,-179.187,5.787,148.784
C06238=1197.376,59.430,-47.221,-179.185,5.787,148.784
C06239=1197.371,59.680,-47.238,-179.182,5.788,148.783
C06240=1197.367,59.929,-47.255,-179.179,5.789,148.782
C06241=1197.362,60.179,-47.270,-179.177,5.789,148.782
C06242=1197.356,60.428,-47.288,-179.174,5.791,148.781
C06243=1197.352,60.678,-47.304,-179.171,5.791,148.781
C06244=1197.347,60.927,-47.321,-179.169,5.792,148.780
C06245=1197.342,61.176,-47.338,-179.167,5.793,148.779
C06246=1197.336,61.425,-47.354,-179.164,5.793,148.779
C06247=1197.332,61.675,-47.371,-179.161,5.795,148.778
C06248=1197.328,61.924,-47.388,-179.159,5.796,148.778
C06249=1197.321,62.174,-47.404,-179.156,5.796,148.777
C06250=1197.317,62.423,-47.420,-179.154,5.797,148.777
C06251=1197.312,62.673,-47.437,-179.151,5.798,148.776
C06252=1197.307,62.922,-47.454,-179.148,5.799,148.775
C06253=1197.302,63.171,-47.471,-179.146,5.800,148.775
C06254=1197.298,63.421,-47.487,-179.143,5.800,148.774
C06255=1197.292,63.670,-47.504,-179.141,5.801,148.773
C06256=1197.287,63.919,-47.521,-179.138,5.803,148.773
C06257=1197.283,64.169,-47.538,-179.135,5.803,148.772
C06258=1197.278,64.419,-47.555,-179.133,5.804,148.772
C06259=1197.273,64.667,-47.571,-179.130,5.805,148.771
C06260=1197.268,64.917,-47.588,-179.128,5.805,148.771
C06261=1197.263,65.167,-47.605,-179.125,5.807,148.770
C06262=1197.258,65.416,-47.621,-179.122,5.807,148.770
C06263=1197.253,65.665,-47.639,-179.120,5.808,148.769
C06264=1197.248,65.915,-47.655,-179.118,5.809,148.768
C06265=1197.244,66.164,-47.672,-179.115,5.809,148.768
C06266=1197.238,66.413,-47.689,-179.112,5.811,148.767
C06267=1197.233,66.663,-47.705,-179.110,5.812,148.767
C06268=1197.228,66.912,-47.723,-179.107,5.812,148.766
C06269=1197.224,67.162,-47.740,-179.104,5.813,148.765
C06270=1197.218,67.411,-47.757,-179.102,5.815,148.765
C06271=1197.214,67.660,-47.774,-179.099,5.815,148.764
C06272=1197.209,67.910,-47.790,-179.096,5.816,148.764
C06273=1197.204,68.159,-47.808,-179.094,5.817,148.763
C06274=1197.199,68.408,-47.824,-179.091,5.818,148.763
C06275=1197.194,68.658,-47.841,-179.089,5.819,148.762
C06276=1197.189,68.907,-47.859,-179.086,5.819,148.761
C06277=1197.184,69.157,-47.876,-179.084,5.820,148.761
C06278=1197.179,69.405,-47.892,-179.081,5.822,148.760
C06279=1197.174,69.655,-47.909,-179.078,5.822,148.760
C06280=1197.169,69.905,-47.926,-179.076,5.823,148.759
C06281=1197.164,70.155,-47.943,-179.074,5.824,148.759
C06282=1197.160,70.403,-47.961,-179.070,5.825,148.758
C06283=1197.154,70.652,-47.978,-179.068,5.826,148.757
C06284=1197.150,70.902,-47.994,-179.066,5.826,148.757
C06285=1197.145,71.152,-48.012,-179.063,5.827,148.756
C06286=1197.140,71.401,-48.029,-179.060,5.829,148.756
C06287=1197.135,71.650,-48.046,-179.058,5.829,148.755
C06288=1197.130,71.899,-48.063,-179.055,5.830,148.754
C06289=1197.125,72.149,-48.080,-179.053,5.831,148.754
C06290=1197.120,72.398,-48.098,-179.050,5.832,148.753
C06291=1197.115,72.648,-48.114,-179.047,5.833,148.753
C06292=1197.110,72.897,-48.132,-179.045,5.834,148.752
C06293=1197.106,73.146,-48.149,-179.042,5.834,148.752
C06294=1197.101,73.396,-48.166,-179.040,5.836,148.751
C06295=1197.096,73.645,-48.183,-179.037,5.836,148.751
C06296=1197.091,73.894,-48.201,-179.034,5.837,148.750
C06297=1197.086,74.144,-48.218,-179.032,5.838,148.749
C06298=1197.081,74.393,-48.235,-179.029,5.839,148.749
C06299=1197.076,74.643,-48.253,-179.027,5.840,148.748
C06300=1197.071,74.892,-48.270,-179.024,5.841,148.748
C06301=1197.067,75.142,-48.286,-179.022,5.841,148.747
C06302=1197.061,75.390,-48.304,-179.019,5.843,148.747
C06303=1197.057,75.640,-48.321,-179.016,5.843,148.746
C06304=1197.052,75.889,-48.339,-179.014,5.844,148.746
C06305=1197.046,76.139,-48.356,-179.011,5.846,148.745
C06306=1197.042,76.388,-48.373,-179.008,5.846,148.744
C06307=1197.037,76.637,-48.391,-179.006,5.847,148.744
C06308=1197.032,76.887,-48.408,-179.003,5.848,148.743
C06309=1197.028,77.136,-48.425,-179.001,5.849,148.743
C06310=1197.022,77.386,-48.443,-178.998,5.850,148.742
C06311=1197.018,77.635,-48.461,-178.995,5.851,148.741
C06312=1197.012,77.884,-48.477,-178.993,5.852,148.741
C06313=1197.008,78.133,-48.495,-178.990,5.853,148.740
C06314=1197.002,78.383,-48.512,-178.988,5.854,148.740
C06315=1196.997,78.632,-48.530,-178.985,5.855,148.739
C06316=1196.993,78.881,-48.547,-178.982,5.856,148.739
C06317=1196.988,79.131,-48.565,-178.980,5.857,148.738
C06318=1196.983,79.380,-48.582,-178.977,5.857,148.737
C06319=1196.978,79.630,-48.600,-178.975,5.859,148.737
C06320=1196.974,79.878,-48.617,-178.972,5.859,148.736
C06321=1196.968,80.128,-48.635,-178.970,5.860,148.736
C06322=1196.964,80.377,-48.653,-178.967,5.862,148.735
C06323=1196.958,80.646,-48.671,-178.964,5.862,148.735
C06324=1196.953,80.914,-48.690,-178.961,5.864,148.734
C06325=1196.947,81.183,-48.709,-178.959,5.865,148.734
C06326=1196.943,81.451,-48.728,-178.956,5.866,148.733
C06327=1196.938,81.700,-48.745,-178.953,5.867,148.732
C06328=1196.933,81.950,-48.763,-178.951,5.867,148.732
C06329=1196.928,82.199,-48.781,-178.948,5.869,148.731
C06330=1196.923,82.449,-48.798,-178.945,5.870,148.731
C06331=1196.918,82.697,-48.816,-178.943,5.870,148.730
C06332=1196.913,82.947,-48.834,-178.940,5.871,148.729
C06333=1196.908,83.196,-48.851,-178.937,5.873,148.729
C06334=1196.903,83.446,-48.869,-178.935,5.873,148.728
C06335=1196.898,83.695,-48.887,-178.933,5.874,148.728
C06336=1196.893,83.945,-48.904,-178.929,5.875,148.727
C06337=1196.888,84.194,-48.922,-178.927,5.876,148.727
C06338=1196.884,84.443,-48.940,-178.925,5.877,148.726
C06339=1196.879,84.692,-48.958,-178.922,5.878,148.726
C06340=1196.874,84.942,-48.975,-178.919,5.879,148.725
C06341=1196.869,85.191,-48.993,-178.917,5.880,148.725
C06342=1196.864,85.440,-49.011,-178.914,5.882,148.724
C06343=1196.859,85.689,-49.029,-178.911,5.882,148.723
C06344=1196.854,85.939,-49.046,-178.909,5.883,148.723
C06345=1196.849,86.188,-49.064,-178.906,5.884,148.722
C06346=1196.845,86.438,-49.082,-178.904,5.885,148.722
C06347=1196.840,86.687,-49.100,-178.901,5.886,148.721
C06348=1196.836,86.936,-49.118,-178.898,5.887,148.721
C06349=1196.830,87.186,-49.135,-178.896,5.888,148.720
C06350=1196.826,87.435,-49.153,-178.893,5.889,148.720
C06351=1196.821,87.684,-49.171,-178.891,5.890,148.719
C06352=1196.816,87.933,-49.189,-178.888,5.891,148.719
C06353=1196.811,88.182,-49.207,-178.885,5.893,148.718
C06354=1196.806,88.432,-49.225,-178.883,5.893,148.717
C06355=1196.801,88.681,-49.243,-178.881,5.894,148.717
C06356=1196.796,88.930,-49.261,-178.877,5.896,148.716
C06357=1196.791,89.180,-49.278,-178.875,5.896,148.716
C06358=1196.787,89.430,-49.296,-178.873,5.897,148.715
C06359=1196.782,89.679,-49.314,-178.869,5.898,148.715
C06360=1196.777,89.928,-49.332,-178.867,5.899,148.714
C06361=1196.772,90.177,-49.350,-178.865,5.900,148.714
C06362=1196.767,90.426,-49.368,-178.862,5.902,148.713
C06363=1196.762,90.676,-49.386,-178.859,5.902,148.713
C06364=1196.757,90.925,-49.404,-178.857,5.904,148.712
C06365=1196.752,91.174,-49.422,-178.854,5.905,148.711
C06366=1196.748,91.424,-49.441,-178.852,5.905,148.711
C06367=1196.742,91.673,-49.459,-178.849,5.907,148.710
C06368=1196.737,91.922,-49.477,-178.847,5.908,148.710
C06369=1196.732,92.172,-49.495,-178.844,5.908,148.709
C06370=1196.727,92.421,-49.513,-178.841,5.910,148.709
C06371=1196.723,92.670,-49.531,-178.839,5.911,148.708
C06372=1196.718,92.920,-49.549,-178.835,5.912,148.708
C06373=1196.713,93.169,-49.567,-178.833,5.913,148.707
C06374=1196.708,93.418,-49.585,-178.831,5.914,148.707
C06375=1196.704,93.667,-49.603,-178.828,5.915,148.706
C06376=1196.699,93.917,-49.621,-178.825,5.916,148.705
C06377=1196.695,94.166,-49.640,-178.823,5.917,148.705
C06378=1196.689,94.415,-49.659,-178.820,5.918,148.704
C06379=1196.684,94.664,-49.677,-178.818,5.919,148.704
C06380=1196.679,94.914,-49.695,-178.815,5.920,148.703
C06381=1196.674,95.163,-49.713,-178.813,5.921,148.703
C06382=1196.670,95.413,-49.731,-178.810,5.922,148.702
C06383=1196.665,95.662,-49.749,-178.807,5.924,148.702
C06384=1196.659,95.911,-49.768,-178.805,5.924,148.701
C06385=1196.655,96.160,-49.787,-178.802,5.926,148.701
C06386=1196.650,96.409,-49.805,-178.799,5.927,148.700
C06387=1196.646,96.659,-49.823,-178.797,5.928,148.700
C06388=1196.641,96.908,-49.841,-178.794,5.929,148.699
C06389=1196.636,97.157,-49.859,-178.792,5.930,148.699
C06390=1196.630,97.406,-49.878,-178.789,5.931,148.698
C06391=1196.626,97.656,-49.896,-178.786,5.932,148.698
C06392=1196.621,97.905,-49.914,-178.784,5.933,148.697
C06393=1196.616,98.154,-49.932,-178.781,5.934,148.697
C06394=1196.611,98.403,-49.952,-178.779,5.935,148.696
C06395=1196.607,98.653,-49.970,-178.776,5.937,148.696
C06396=1196.602,98.902,-49.988,-178.773,5.937,148.695
C06397=1196.597,99.152,-50.006,-178.770,5.939,148.694
C06398=1196.592,99.401,-50.026,-178.768,5.940,148.694
C06399=1196.587,99.650,-50.044,-178.766,5.941,148.693
C06400=1196.582,99.899,-50.062,-178.763,5.942,148.693
C06401=1196.578,100.148,-50.080,-178.760,5.943,148.692
C06402=1196.573,100.398,-50.099,-178.757,5.944,148.692
C06403=1196.568,100.647,-50.117,-178.755,5.945,148.691
C06404=1196.563,100.896,-50.136,-178.752,5.947,148.691
C06405=1196.558,101.146,-50.155,-178.750,5.948,148.690
C06406=1196.553,101.395,-50.173,-178.747,5.948,148.690
C06407=1196.548,101.644,-50.192,-178.744,5.950,148.689
C06408=1196.543,101.894,-50.211,-178.742,5.950,148.689
C06409=1196.539,102.143,-50.229,-178.739,5.952,148.688
C06410=1196.534,102.392,-50.247,-178.737,5.953,148.687
C06411=1196.529,102.642,-50.266,-178.734,5.954,148.687
C06412=1196.524,102.891,-50.285,-178.731,5.955,148.686
C06413=1196.519,103.140,-50.303,-178.729,5.956,148.686
C06414=1196.515,103.389,-50.322,-178.726,5.958,148.686
C06415=1196.510,103.638,-50.340,-178.724,5.958,148.685
C06416=1196.505,103.887,-50.359,-178.721,5.960,148.685
C06417=1196.500,104.137,-50.378,-178.718,5.961,148.684
C06418=1196.495,104.386,-50.397,-178.716,5.962,148.684
C06419=1196.490,104.635,-50.415,-178.713,5.963,148.683
C06420=1196.486,104.884,-50.434,-178.710,5.965,148.682
C06421=1196.481,105.134,-50.452,-178.708,5.965,148.682
C06422=1196.476,105.383,-50.472,-178.706,5.966,148.681
C06423=1196.471,105.632,-50.490,-178.702,5.968,148.681
C06424=1196.466,105.881,-50.509,-178.700,5.969,148.680
C06425=1196.461,106.131,-50.528,-178.697,5.970,148.680
C06426=1196.456,106.380,-50.547,-178.695,5.971,148.679
C06427=1196.452,106.649,-50.567,-178.692,5.972,148.679
C06428=1196.446,106.917,-50.587,-178.689,5.974,148.678
C06429=1196.440,107.185,-50.607,-178.687,5.975,148.678
C06430=1196.436,107.454,-50.628,-178.683,5.976,148.677
C06431=1196.431,107.703,-50.647,-178.681,5.977,148.677
C06432=1196.426,107.952,-50.665,-178.678,5.978,148.676
C06433=1196.421,108.201,-50.685,-178.676,5.979,148.676
C06434=1196.416,108.451,-50.703,-178.673,5.981,148.675
C06435=1196.412,108.700,-50.723,-178.671,5.982,148.674
C06436=1196.407,108.949,-50.741,-178.668,5.983,148.674
C06437=1196.402,109.199,-50.760,-178.665,5.984,148.673
C06438=1196.397,109.447,-50.779,-178.663,5.986,148.673
C06439=1196.392,109.697,-50.799,-178.660,5.986,148.672
C06440=1196.388,109.946,-50.816,-178.657,5.988,148.672
C06441=1196.383,110.196,-50.836,-178.655,5.989,148.671
C06442=1196.378,110.444,-50.855,-178.652,5.990,148.671
C06443=1196.373,110.693,-50.874,-178.650,5.991,148.671
C06444=1196.368,110.943,-50.893,-178.647,5.993,148.670
C06445=1196.363,111.192,-50.912,-178.644,5.994,148.669
C06446=1196.358,111.442,-50.931,-178.641,5.995,148.669
C06447=1196.354,111.690,-50.950,-178.639,5.996,148.668
C06448=1196.349,111.940,-50.969,-178.636,5.997,148.668
C06449=1196.343,112.189,-50.988,-178.634,5.998,148.667
C06450=1196.339,112.438,-51.007,-178.631,6.000,148.667
C06451=1196.334,112.687,-51.027,-178.629,6.001,148.666
C06452=1196.330,112.937,-51.046,-178.626,6.002,148.666
C06453=1196.325,113.185,-51.065,-178.623,6.003,148.665
C06454=1196.320,113.436,-51.084,-178.621,6.005,148.665
C06455=1196.315,113.684,-51.103,-178.618,6.006,148.665
C06456=1196.310,113.934,-51.122,-178.615,6.007,148.664
C06457=1196.306,114.183,-51.142,-178.613,6.008,148.663
C06458=1196.301,114.432,-51.161,-178.610,6.009,148.663
C06459=1196.296,114.681,-51.180,-178.608,6.010,148.662
C06460=1196.291,114.930,-51.200,-178.605,6.012,148.662
C06461=1196.287,115.180,-51.218,-178.602,6.013,148.661
C06462=1196.281,115.429,-51.237,-178.600,6.014,148.661
C06463=1196.277,115.679,-51.257,-178.597,6.015,148.660
C06464=1196.271,115.927,-51.276,-178.594,6.017,148.660
C06465=1196.267,116.177,-51.295,-178.592,6.017,148.659
C06466=1196.262,116.426,-51.315,-178.589,6.019,148.659
C06467=1196.257,116.675,-51.334,-178.587,6.020,148.659
C06468=1196.253,116.924,-51.353,-178.584,6.021,148.658
C06469=1196.248,117.173,-51.373,-178.582,6.022,148.657
C06470=1196.243,117.423,-51.392,-178.579,6.024,148.657
C06471=1196.238,117.672,-51.412,-178.576,6.026,148.656
C06472=1196.234,117.921,-51.431,-178.574,6.026,148.656
C06473=1196.229,118.171,-51.450,-178.571,6.028,148.655
C06474=1196.224,118.419,-51.470,-178.568,6.029,148.655
C06475=1196.219,118.669,-51.489,-178.565,6.030,148.654
C06476=1196.214,118.918,-51.508,-178.563,6.031,148.654
C06477=1196.210,119.167,-51.528,-178.560,6.033,148.654
C06478=1196.205,119.417,-51.547,-178.558,6.033,148.653
C06479=1196.200,119.665,-51.567,-178.555,6.035,148.653
C06480=1196.195,119.914,-51.587,-178.553,6.036,148.652
C06481=1196.190,120.164,-51.607,-178.550,6.038,148.652
C06482=1196.186,120.413,-51.625,-178.547,6.039,148.651
C06483=1196.181,120.662,-51.645,-178.545,6.040,148.650
C06484=1196.176,120.912,-51.665,-178.542,6.042,148.650
C06485=1196.171,121.161,-51.684,-178.540,6.043,148.650
C06486=1196.166,121.410,-51.703,-178.537,6.044,148.649
C06487=1196.162,121.659,-51.724,-178.534,6.045,148.649
C06488=1196.157,121.908,-51.743,-178.531,6.046,148.648
C06489=1196.152,122.157,-51.762,-178.529,6.047,148.648
C06490=1196.148,122.407,-51.782,-178.526,6.049,148.647
C06491=1196.142,122.656,-51.801,-178.523,6.051,148.647
C06492=1196.138,122.905,-51.822,-178.521,6.051,148.646
C06493=1196.133,123.154,-51.841,-178.518,6.053,148.646
C06494=1196.128,123.403,-51.860,-178.516,6.054,148.645
C06495=1196.123,123.653,-51.880,-178.513,6.056,148.645
C06496=1196.118,123.902,-51.900,-178.511,6.056,148.644
C06497=1196.113,124.150,-51.920,-178.508,6.058,148.644
C06498=1196.109,124.400,-51.939,-178.505,6.060,148.643
C06499=1196.104,124.649,-51.959,-178.502,6.060,148.643
C06500=1196.100,124.898,-51.979,-178.500,6.062,148.642
C06501=1196.095,125.147,-51.998,-178.498,6.063,148.642
C06502=1196.090,125.397,-52.018,-178.494,6.064,148.641
C06503=1196.085,125.646,-52.038,-178.492,6.065,148.641
C06504=1196.081,125.895,-52.058,-178.490,6.067,148.640
C06505=1196.075,126.144,-52.077,-178.487,6.068,148.640
C06506=1196.071,126.393,-52.098,-178.484,6.069,148.639
C06507=1196.066,126.643,-52.117,-178.482,6.071,148.639
C06508=1196.061,126.892,-52.137,-178.479,6.072,148.638
C06509=1196.056,127.140,-52.157,-178.476,6.074,148.638
C06510=1196.052,127.390,-52.176,-178.474,6.075,148.638
C06511=1196.047,127.639,-52.197,-178.471,6.076,148.637
C06512=1196.042,127.888,-52.217,-178.468,6.078,148.637
C06513=1196.037,128.137,-52.236,-178.466,6.079,148.636
C06514=1196.033,128.386,-52.256,-178.463,6.080,148.636
C06515=1196.028,128.636,-52.276,-178.460,6.082,148.635
C06516=1196.024,128.885,-52.296,-178.458,6.083,148.635
C06517=1196.019,129.134,-52.316,-178.455,6.084,148.634
C06518=1196.013,129.383,-52.336,-178.453,6.085,148.634
C06519=1196.008,129.632,-52.356,-178.450,6.087,148.633
C06520=1196.004,129.881,-52.376,-178.447,6.088,148.633
C06521=1195.999,130.131,-52.396,-178.445,6.089,148.632
C06522=1195.995,130.380,-52.417,-178.442,6.091,148.632
C06523=1195.989,130.629,-52.436,-178.440,6.092,148.631
C06524=1195.985,130.878,-52.456,-178.437,6.093,148.631
C06525=1195.980,131.127,-52.476,-178.434,6.095,148.631
C06526=1195.976,131.376,-52.496,-178.432,6.096,148.630
C06527=1195.970,131.626,-52.516,-178.429,6.097,148.630
C06528=1195.966,131.875,-52.537,-178.426,6.099,148.629
C06529=1195.961,132.123,-52.557,-178.424,6.100,148.629
C06530=1195.956,132.373,-52.576,-178.421,6.102,148.628
C06531=1195.951,132.641,-52.599,-178.418,6.103,148.628
C06532=1195.946,132.910,-52.620,-178.415,6.105,148.627
C06533=1195.940,133.179,-52.642,-178.413,6.106,148.627
C06534=1195.936,133.448,-52.664,-178.410,6.107,148.626
C06535=1195.931,133.696,-52.683,-178.407,6.109,148.626
C06536=1195.926,133.946,-52.704,-178.405,6.110,148.625
C06537=1195.921,134.195,-52.724,-178.402,6.111,148.625
C06538=1195.916,134.444,-52.744,-178.399,6.113,148.624
C06539=1195.912,134.693,-52.764,-178.397,6.114,148.624
C06540=1195.907,134.942,-52.785,-178.394,6.115,148.623
C06541=1195.902,135.191,-52.806,-178.391,6.117,148.623
C06542=1195.898,135.441,-52.825,-178.389,6.118,148.623
C06543=1195.893,135.690,-52.846,-178.386,6.120,148.622
C06544=1195.889,135.939,-52.866,-178.383,6.121,148.622
C06545=1195.883,136.188,-52.886,-178.381,6.122,148.621
C06546=1195.878,136.437,-52.906,-178.378,6.124,148.621
C06547=1195.874,136.686,-52.927,-178.375,6.126,148.620
C06548=1195.869,136.935,-52.947,-178.373,6.126,148.620
C06549=1195.864,137.184,-52.968,-178.370,6.128,148.619
C06550=1195.859,137.434,-52.988,-178.367,6.130,148.619
C06551=1195.855,137.683,-53.008,-178.365,6.131,148.618
C06552=1195.850,137.932,-53.029,-178.363,6.132,148.618
C06553=1195.845,138.181,-53.050,-178.360,6.134,148.618
C06554=1195.841,138.430,-53.070,-178.357,6.135,148.617
C06555=1195.836,138.679,-53.091,-178.355,6.137,148.617
C06556=1195.831,138.929,-53.111,-178.352,6.138,148.616
C06557=1195.827,139.178,-53.131,-178.350,6.139,148.616
C06558=1195.821,139.427,-53.152,-178.347,6.141,148.615
C06559=1195.817,139.676,-53.172,-178.344,6.142,148.615
C06560=1195.812,139.925,-53.193,-178.342,6.143,148.614
C06561=1195.807,140.174,-53.214,-178.339,6.145,148.614
C06562=1195.803,140.423,-53.234,-178.336,6.147,148.613
C06563=1195.798,140.672,-53.255,-178.334,6.148,148.613
C06564=1195.793,140.921,-53.275,-178.331,6.149,148.613
C06565=1195.789,141.170,-53.296,-178.328,6.151,148.612
C06566=1195.784,141.419,-53.317,-178.326,6.152,148.612
C06567=1195.779,141.668,-53.337,-178.323,6.153,148.611
C06568=1195.774,141.918,-53.358,-178.320,6.155,148.611
C06569=1195.770,142.167,-53.378,-178.318,6.156,148.610
C06570=1195.765,142.415,-53.399,-178.315,6.158,148.610
C06571=1195.760,142.665,-53.420,-178.312,6.159,148.609
C06572=1195.756,142.914,-53.440,-178.310,6.161,148.609
C06573=1195.750,143.163,-53.461,-178.307,6.162,148.608
C06574=1195.746,143.412,-53.481,-178.305,6.164,148.608
C06575=1195.741,143.661,-53.502,-178.302,6.165,148.608
C06576=1195.736,143.910,-53.523,-178.300,6.166,148.607
C06577=1195.731,144.159,-53.544,-178.297,6.168,148.607
C06578=1195.727,144.408,-53.564,-178.294,6.169,148.606
C06579=1195.722,144.658,-53.585,-178.292,6.170,148.606
C06580=1195.717,144.907,-53.605,-178.289,6.172,148.605
C06581=1195.713,145.156,-53.627,-178.286,6.174,148.605
C06582=1195.708,145.405,-53.647,-178.283,6.175,148.604
C06583=1195.703,145.654,-53.669,-178.281,6.176,148.604
C06584=1195.699,145.903,-53.689,-178.278,6.178,148.604
C06585=1195.694,146.152,-53.710,-178.276,6.180,148.603
C06586=1195.689,146.401,-53.731,-178.273,6.181,148.603
C06587=1195.684,146.650,-53.751,-178.270,6.182,148.602
C06588=1195.680,146.899,-53.772,-178.268,6.184,148.602
C06589=1195.675,147.148,-53.794,-178.265,6.186,148.602
C06590=1195.670,147.397,-53.814,-178.262,6.186,148.601
C06591=1195.666,147.647,-53.835,-178.260,6.188,148.601
C06592=1195.660,147.896,-53.856,-178.257,6.190,148.600
C06593=1195.656,148.145,-53.877,-178.254,6.192,148.600
C06594=1195.651,148.394,-53.898,-178.252,6.193,148.599
C06595=1195.647,148.643,-53.919,-178.249,6.194,148.599
C06596=1195.642,148.892,-53.940,-178.246,6.196,148.598
C06597=1195.637,149.141,-53.961,-178.244,6.197,148.598
C06598=1195.633,149.390,-53.982,-178.242,6.199,148.598
C06599=1195.628,149.640,-54.003,-178.239,6.200,148.597
C06600=1195.623,149.888,-54.025,-178.236,6.202,148.597
C06601=1195.618,150.137,-54.045,-178.234,6.203,148.596
C06602=1195.613,150.386,-54.066,-178.231,6.205,148.596
C06603=1195.608,150.635,-54.088,-178.228,6.206,148.596
C06604=1195.605,150.885,-54.108,-178.225,6.208,148.595
C06605=1195.599,151.134,-54.129,-178.223,6.209,148.595
C06606=1195.594,151.383,-54.151,-178.220,6.211,148.594
C06607=1195.590,151.632,-54.171,-178.218,6.212,148.594
C06608=1195.585,151.881,-54.192,-178.215,6.214,148.593
C06609=1195.581,152.130,-54.214,-178.212,6.215,148.593
C06610=1195.575,152.379,-54.235,-178.210,6.217,148.592
C06611=1195.571,152.628,-54.257,-178.207,6.218,148.592
C06612=1195.566,152.877,-54.277,-178.204,6.220,148.592
C06613=1195.561,153.126,-54.299,-178.202,6.221,148.591
C06614=1195.557,153.375,-54.320,-178.200,6.223,148.591
C06615=1195.553,153.624,-54.342,-178.196,6.224,148.590
C06616=1195.547,153.873,-54.363,-178.194,6.226,148.590
C06617=1195.542,154.122,-54.384,-178.191,6.228,148.590
C06618=1195.538,154.372,-54.406,-178.189,6.229,148.589
C06619=1195.534,154.620,-54.427,-178.186,6.231,148.589
C06620=1195.529,154.869,-54.448,-178.184,6.232,148.588
C06621=1195.524,155.118,-54.469,-178.180,6.234,148.588
C06622=1195.519,155.368,-54.491,-178.178,6.235,148.587
C06623=1195.514,155.617,-54.512,-178.176,6.237,148.587
C06624=1195.510,155.866,-54.533,-178.173,6.238,148.587
C06625=1195.505,156.114,-54.554,-178.170,6.240,148.586
C06626=1195.500,156.364,-54.576,-178.167,6.242,148.586
C06627=1195.496,156.613,-54.597,-178.165,6.243,148.585
C06628=1195.491,156.861,-54.619,-178.162,6.244,148.585
C06629=1195.486,157.111,-54.640,-178.160,6.246,148.585
C06630=1195.482,157.360,-54.662,-178.157,6.248,148.584
C06631=1195.477,157.608,-54.683,-178.155,6.249,148.584
C06632=1195.472,157.858,-54.704,-178.152,6.251,148.583
C06633=1195.468,158.107,-54.726,-178.149,6.252,148.583
C06634=1195.463,158.356,-54.748,-178.146,6.254,148.582
C06635=1195.458,158.625,-54.771,-178.144,6.256,148.582
C06636=1195.453,158.894,-54.794,-178.141,6.257,148.582
C06637=1195.448,159.163,-54.817,-178.138,6.259,148.581
C06638=1195.443,159.432,-54.841,-178.135,6.261,148.581
C06639=1195.437,159.681,-54.862,-178.133,6.262,148.580
C06640=1195.433,159.930,-54.884,-178.130,6.264,148.580
C06641=1195.428,160.179,-54.906,-178.128,6.265,148.580
C06642=1195.423,160.428,-54.927,-178.125,6.267,148.579
C06643=1195.419,160.678,-54.949,-178.122,6.268,148.579
C06644=1195.414,160.926,-54.970,-178.119,6.270,148.578
C06645=1195.409,161.175,-54.992,-178.117,6.272,148.578
C06646=1195.405,161.424,-55.014,-178.114,6.273,148.577
C06647=1195.400,161.673,-55.036,-178.112,6.275,148.577
C06648=1195.395,161.923,-55.057,-178.109,6.276,148.577
C06649=1195.391,162.172,-55.079,-178.106,6.278,148.576
C06650=1195.386,162.420,-55.100,-178.103,6.280,148.576
C06651=1195.381,162.670,-55.122,-178.101,6.282,148.575
C06652=1195.377,162.918,-55.144,-178.099,6.282,148.575
C06653=1195.372,163.168,-55.166,-178.096,6.284,148.575
C06654=1195.367,163.416,-55.188,-178.093,6.286,148.574
C06655=1195.362,163.665,-55.209,-178.090,6.288,148.574
C06656=1195.358,163.915,-55.231,-178.088,6.290,148.574
C06657=1195.353,164.163,-55.253,-178.085,6.291,148.573
C06658=1195.349,164.413,-55.275,-178.083,6.292,148.573
C06659=1195.344,164.661,-55.296,-178.080,6.294,148.572
C06660=1195.340,164.911,-55.318,-178.077,6.296,148.572
C06661=1195.335,165.159,-55.340,-178.075,6.297,148.571
C06662=1195.330,165.408,-55.362,-178.072,6.299,148.571
C06663=1195.326,165.657,-55.384,-178.069,6.301,148.571
C06664=1195.321,165.906,-55.405,-178.067,6.303,148.570
C06665=1195.317,166.155,-55.427,-178.064,6.304,148.570
C06666=1195.312,166.404,-55.449,-178.062,6.306,148.570
C06667=1195.307,166.654,-55.472,-178.059,6.307,148.569
C06668=1195.302,166.902,-55.493,-178.056,6.309,148.569
C06669=1195.298,167.152,-55.515,-178.053,6.311,148.568
C06670=1195.293,167.400,-55.537,-178.051,6.312,148.568
C06671=1195.288,167.650,-55.559,-178.048,6.313,148.568
C06672=1195.284,167.898,-55.581,-178.046,6.315,148.567
C06673=1195.279,168.148,-55.603,-178.043,6.317,148.567
C06674=1195.274,168.396,-55.626,-178.040,6.319,148.566
C06675=1195.270,168.645,-55.648,-178.038,6.320,148.566
C06676=1195.265,168.894,-55.670,-178.035,6.322,148.566
C06677=1195.261,169.143,-55.692,-178.032,6.324,148.565
C06678=1195.256,169.392,-55.713,-178.030,6.326,148.565
C06679=1195.251,169.642,-55.736,-178.027,6.326,148.564
C06680=1195.246,169.890,-55.758,-178.024,6.328,148.564
C06681=1195.242,170.139,-55.780,-178.022,6.330,148.564
C06682=1195.237,170.388,-55.802,-178.019,6.332,148.563
C06683=1195.232,170.637,-55.825,-178.016,6.334,148.563
C06684=1195.227,170.886,-55.846,-178.014,6.335,148.563
C06685=1195.223,171.135,-55.869,-178.011,6.337,148.562
C06686=1195.218,171.383,-55.891,-178.008,6.339,148.562
C06687=1195.213,171.633,-55.914,-178.006,6.340,148.561
C06688=1195.209,171.882,-55.936,-178.004,6.342,148.561
C06689=1195.204,172.131,-55.957,-178.001,6.344,148.561
C06690=1195.199,172.380,-55.981,-177.998,6.345,148.560
C06691=1195.195,172.628,-56.002,-177.996,6.347,148.560
C06692=1195.190,172.878,-56.024,-177.993,6.349,148.560
C06693=1195.186,173.126,-56.047,-177.990,6.351,148.559
C06694=1195.181,173.375,-56.069,-177.988,6.353,148.559
C06695=1195.176,173.625,-56.091,-177.985,6.354,148.558
C06696=1195.172,173.873,-56.113,-177.982,6.356,148.558
C06697=1195.167,174.123,-56.137,-177.980,6.357,148.558
C06698=1195.162,174.371,-56.158,-177.977,6.359,148.557
C06699=1195.157,174.620,-56.182,-177.974,6.360,148.557
C06700=1195.153,174.870,-56.204,-177.972,6.362,148.556
C06701=1195.148,175.118,-56.225,-177.969,6.364,148.556
C06702=1195.143,175.367,-56.249,-177.966,6.366,148.556
C06703=1195.139,175.617,-56.271,-177.964,6.368,148.555
C06704=1195.135,175.865,-56.293,-177.961,6.369,148.555
C06705=1195.130,176.114,-56.316,-177.958,6.371,148.555
C06706=1195.125,176.363,-56.337,-177.956,6.373,148.554
C06707=1195.120,176.612,-56.361,-177.953,6.375,148.554
C06708=1195.116,176.861,-56.383,-177.950,6.376,148.554
C06709=1195.111,177.110,-56.406,-177.948,6.377,148.553
C06710=1195.106,177.359,-56.428,-177.946,6.379,148.553
C06711=1195.102,177.608,-56.451,-177.943,6.381,148.552
C06712=1195.097,177.857,-56.473,-177.940,6.383,148.552
C06713=1195.093,178.105,-56.496,-177.938,6.385,148.552
C06714=1195.088,178.355,-56.518,-177.935,6.386,148.551
C06715=1195.083,178.603,-56.541,-177.932,6.388,148.551
C06716=1195.078,178.852,-56.564,-177.930,6.390,148.551
C06717=1195.074,179.101,-56.586,-177.927,6.392,148.550
C06718=1195.069,179.350,-56.610,-177.924,6.394,148.550
C06719=1195.065,179.599,-56.631,-177.922,6.395,148.550
C06720=1195.060,179.848,-56.655,-177.919,6.397,148.549
C06721=1195.056,180.097,-56.677,-177.916,6.399,148.549
C06722=1195.050,180.346,-56.700,-177.914,6.401,148.549
C06723=1195.046,180.594,-56.722,-177.911,6.403,148.548
C06724=1195.041,180.844,-56.745,-177.908,6.404,148.548
C06725=1195.037,181.093,-56.768,-177.906,6.405,148.547
C06726=1195.032,181.341,-56.791,-177.904,6.407,148.547
C06727=1195.028,181.590,-56.813,-177.901,6.409,148.547
C06728=1195.023,181.840,-56.836,-177.898,6.411,148.546
C06729=1195.018,182.089,-56.860,-177.896,6.413,148.546
C06730=1195.014,182.337,-56.881,-177.893,6.414,148.546
C06731=1195.009,182.586,-56.905,-177.890,6.416,148.545
C06732=1195.005,182.835,-56.927,-177.888,6.418,148.545
C06733=1195.000,183.084,-56.951,-177.885,6.420,148.545
C06734=1194.995,183.334,-56.973,-177.882,6.422,148.544
C06735=1194.991,183.582,-56.996,-177.880,6.423,148.544
C06736=1194.986,183.831,-57.019,-177.877,6.425,148.543
C06737=1194.982,184.079,-57.042,-177.874,6.427,148.543
C06738=1194.977,184.329,-57.064,-177.872,6.429,148.543
C06739=1194.972,184.598,-57.090,-177.869,6.431,148.542
C06740=1194.967,184.868,-57.115,-177.866,6.432,148.542
C06741=1194.962,185.137,-57.140,-177.863,6.435,148.542
C06742=1194.957,185.407,-57.165,-177.860,6.436,148.541
C06743=1194.952,185.655,-57.187,-177.857,6.438,148.541
C06744=1194.947,185.904,-57.211,-177.855,6.440,148.540
C06745=1194.942,186.154,-57.233,-177.852,6.442,148.540
C06746=1194.939,186.403,-57.256,-177.850,6.444,148.540
C06747=1194.934,186.652,-57.279,-177.847,6.446,148.540
C06748=1194.929,186.901,-57.303,-177.844,6.448,148.539
C06749=1194.925,187.149,-57.325,-177.842,6.449,148.539
C06750=1194.920,187.398,-57.348,-177.839,6.451,148.539
C06751=1194.915,187.647,-57.372,-177.836,6.453,148.538
C06752=1194.910,187.896,-57.395,-177.834,6.455,148.538
C06753=1194.906,188.144,-57.418,-177.831,6.457,148.538
C06754=1194.902,188.394,-57.441,-177.828,6.458,148.537
C06755=1194.897,188.643,-57.465,-177.826,6.460,148.537
C06756=1194.892,188.892,-57.488,-177.823,6.462,148.536
C06757=1194.887,189.140,-57.511,-177.820,6.464,148.536
C06758=1194.883,189.389,-57.534,-177.818,6.466,148.536
C06759=1194.878,189.638,-57.557,-177.815,6.467,148.535
C06760=1194.874,189.887,-57.580,-177.812,6.469,148.535
C06761=1194.869,190.136,-57.604,-177.810,6.471,148.535
C06762=1194.864,190.385,-57.627,-177.807,6.473,148.534
C06763=1194.860,190.633,-57.650,-177.804,6.475,148.534
C06764=1194.856,190.883,-57.673,-177.802,6.476,148.534
C06765=1194.851,191.132,-57.697,-177.800,6.479,148.534
C06766=1194.846,191.381,-57.720,-177.797,6.480,148.533
C06767=1194.841,191.629,-57.743,-177.794,6.482,148.533
C06768=1194.837,191.877,-57.767,-177.792,6.484,148.532
C06769=1194.832,192.126,-57.790,-177.789,6.486,148.532
C06770=1194.827,192.375,-57.814,-177.786,6.488,148.532
C06771=1194.823,192.624,-57.837,-177.784,6.489,148.531
C06772=1194.819,192.873,-57.860,-177.781,6.491,148.531
C06773=1194.814,193.122,-57.883,-177.778,6.493,148.531
C06774=1194.809,193.371,-57.907,-177.776,6.495,148.530
C06775=1194.805,193.620,-57.931,-177.773,6.497,148.530
C06776=1194.800,193.869,-57.954,-177.770,6.498,148.530
C06777=1194.795,194.118,-57.977,-177.768,6.501,148.530
C06778=1194.791,194.367,-58.001,-177.765,6.502,148.529
C06779=1194.786,194.615,-58.025,-177.763,6.504,148.529
C06780=1194.782,194.864,-58.048,-177.760,6.506,148.528
C06781=1194.777,195.113,-58.072,-177.757,6.508,148.528
C06782=1194.772,195.362,-58.096,-177.755,6.510,148.528
C06783=1194.768,195.611,-58.119,-177.752,6.512,148.527
C06784=1194.763,195.860,-58.142,-177.749,6.514,148.527
C06785=1194.758,196.109,-58.166,-177.746,6.516,148.527
C06786=1194.754,196.357,-58.190,-177.744,6.518,148.526
C06787=1194.749,196.606,-58.213,-177.741,6.520,148.526
C06788=1194.745,196.855,-58.236,-177.739,6.522,148.526
C06789=1194.740,197.104,-58.261,-177.736,6.523,148.526
C06790=1194.735,197.353,-58.284,-177.733,6.525,148.525
C06791=1194.731,197.601,-58.308,-177.731,6.527,148.525
C06792=1194.726,197.850,-58.331,-177.728,6.529,148.525
C06793=1194.722,198.099,-58.355,-177.726,6.531,148.524
C06794=1194.717,198.348,-58.379,-177.723,6.533,148.524
C06795=1194.713,198.597,-58.402,-177.720,6.534,148.524
C06796=1194.708,198.845,-58.426,-177.718,6.536,148.523
C06797=1194.704,199.095,-58.450,-177.715,6.538,148.523
C06798=1194.700,199.343,-58.474,-177.713,6.540,148.523
C06799=1194.695,199.592,-58.497,-177.709,6.543,148.522
C06800=1194.690,199.841,-58.522,-177.707,6.545,148.522
C06801=1194.685,200.090,-58.545,-177.704,6.546,148.522
C06802=1194.681,200.338,-58.569,-177.702,6.548,148.521
C06803=1194.676,200.587,-58.593,-177.699,6.550,148.521
C06804=1194.672,200.836,-58.617,-177.697,6.552,148.521
C06805=1194.667,201.085,-58.640,-177.694,6.554,148.521
C06806=1194.663,201.333,-58.664,-177.691,6.556,148.520
C06807=1194.658,201.582,-58.688,-177.689,6.558,148.520
C06808=1194.653,201.832,-58.713,-177.686,6.559,148.520
C06809=1194.649,202.081,-58.736,-177.683,6.561,148.519
C06810=1194.644,202.329,-58.760,-177.681,6.564,148.519
C06811=1194.640,202.578,-58.784,-177.678,6.566,148.519
C06812=1194.635,202.827,-58.808,-177.675,6.568,148.518
C06813=1194.630,203.075,-58.832,-177.673,6.570,148.518
C06814=1194.626,203.324,-58.856,-177.670,6.571,148.518
C06815=1194.622,203.573,-58.880,-177.667,6.573,148.517
C06816=1194.617,203.822,-58.904,-177.665,6.575,148.517
C06817=1194.613,204.070,-58.928,-177.663,6.577,148.517
C06818=1194.607,204.320,-58.952,-177.660,6.579,148.517
C06819=1194.603,204.568,-58.976,-177.657,6.581,148.516
C06820=1194.599,204.816,-59.000,-177.654,6.583,148.516
C06821=1194.594,205.066,-59.024,-177.651,6.585,148.516
C06822=1194.589,205.315,-59.049,-177.649,6.587,148.515
C06823=1194.585,205.563,-59.073,-177.647,6.589,148.515
C06824=1194.580,205.812,-59.097,-177.644,6.591,148.515
C06825=1194.575,206.061,-59.121,-177.641,6.593,148.514
C06826=1194.571,206.310,-59.145,-177.639,6.595,148.514
C06827=1194.567,206.559,-59.169,-177.636,6.596,148.514
C06828=1194.562,206.807,-59.194,-177.633,6.599,148.513
C06829=1194.557,207.056,-59.218,-177.631,6.601,148.513
C06830=1194.553,207.305,-59.241,-177.628,6.603,148.513
C06831=1194.548,207.554,-59.266,-177.625,6.605,148.513
C06832=1194.544,207.803,-59.291,-177.623,6.607,148.512
C06833=1194.539,208.051,-59.315,-177.620,6.608,148.512
C06834=1194.534,208.300,-59.339,-177.618,6.611,148.512
C06835=1194.530,208.549,-59.364,-177.615,6.612,148.511
C06836=1194.526,208.797,-59.388,-177.612,6.615,148.511
C06837=1194.521,209.046,-59.412,-177.609,6.617,148.511
C06838=1194.516,209.295,-59.436,-177.607,6.619,148.511
C06839=1194.512,209.544,-59.461,-177.604,6.621,148.510
C06840=1194.507,209.793,-59.485,-177.602,6.623,148.510
C06841=1194.503,210.041,-59.509,-177.599,6.625,148.510
C06842=1194.498,210.291,-59.534,-177.596,6.626,148.509
C06843=1194.493,210.561,-59.561,-177.593,6.629,148.509
C06844=1194.488,210.831,-59.587,-177.591,6.631,148.509
C06845=1194.484,211.101,-59.614,-177.587,6.633,148.508
C06846=1194.479,211.372,-59.640,-177.585,6.635,148.508
C06847=1194.474,211.621,-59.665,-177.583,6.637,148.508
C06848=1194.469,211.869,-59.689,-177.579,6.640,148.508
C06849=1194.464,212.118,-59.714,-177.577,6.642,148.507
C06850=1194.461,212.367,-59.739,-177.574,6.644,148.507
C06851=1194.455,212.615,-59.763,-177.572,6.646,148.507
C06852=1194.451,212.864,-59.787,-177.569,6.648,148.507
C06853=1194.447,213.113,-59.812,-177.567,6.649,148.506
C06854=1194.442,213.362,-59.836,-177.563,6.652,148.506
C06855=1194.437,213.610,-59.861,-177.561,6.654,148.506
C06856=1194.433,213.860,-59.885,-177.559,6.656,148.505
C06857=1194.428,214.108,-59.910,-177.556,6.658,148.505
C06858=1194.424,214.357,-59.935,-177.553,6.660,148.505
C06859=1194.419,214.605,-59.960,-177.551,6.662,148.504
C06860=1194.414,214.854,-59.985,-177.548,6.665,148.504
C06861=1194.411,215.103,-60.009,-177.545,6.666,148.504
C06862=1194.405,215.352,-60.034,-177.543,6.668,148.504
C06863=1194.401,215.600,-60.058,-177.540,6.670,148.503
C06864=1194.397,215.849,-60.084,-177.538,6.672,148.503
C06865=1194.392,216.098,-60.108,-177.534,6.675,148.503
C06866=1194.388,216.347,-60.133,-177.532,6.677,148.503
C06867=1194.383,216.596,-60.157,-177.529,6.678,148.502
C06868=1194.379,216.844,-60.182,-177.527,6.681,148.502
C06869=1194.374,217.093,-60.207,-177.524,6.682,148.502
C06870=1194.369,217.342,-60.232,-177.521,6.685,148.502
C06871=1194.365,217.591,-60.256,-177.519,6.687,148.501
C06872=1194.360,217.839,-60.282,-177.516,6.689,148.501
C06873=1194.355,218.088,-60.306,-177.514,6.691,148.501
C06874=1194.351,218.337,-60.331,-177.511,6.693,148.500
C06875=1194.347,218.585,-60.356,-177.508,6.694,148.500
C06876=1194.342,218.834,-60.381,-177.506,6.697,148.500
C06877=1194.338,219.082,-60.406,-177.503,6.699,148.500
C06878=1194.333,219.332,-60.431,-177.500,6.701,148.499
C06879=1194.328,219.580,-60.456,-177.498,6.703,148.499
C06880=1194.325,219.829,-60.481,-177.495,6.706,148.499
C06881=1194.320,220.077,-60.506,-177.492,6.708,148.499
C06882=1194.315,220.326,-60.531,-177.490,6.710,148.498
C06883=1194.310,220.575,-60.556,-177.488,6.712,148.498
C06884=1194.307,220.824,-60.580,-177.485,6.713,148.498
C06885=1194.302,221.072,-60.606,-177.482,6.716,148.498
C06886=1194.297,221.322,-60.631,-177.479,6.718,148.497
C06887=1194.292,221.570,-60.656,-177.477,6.720,148.497
C06888=1194.289,221.819,-60.681,-177.474,6.722,148.497
C06889=1194.284,222.067,-60.706,-177.472,6.724,148.496
C06890=1194.279,222.316,-60.731,-177.469,6.727,148.496
C06891=1194.274,222.565,-60.756,-177.466,6.729,148.496
C06892=1194.270,222.814,-60.781,-177.464,6.730,148.496
C06893=1194.266,223.062,-60.806,-177.461,6.733,148.496
C06894=1194.262,223.311,-60.832,-177.458,6.735,148.495
C06895=1194.256,223.559,-60.857,-177.456,6.737,148.495
C06896=1194.252,223.808,-60.882,-177.453,6.739,148.495
C06897=1194.247,224.057,-60.907,-177.451,6.741,148.494
C06898=1194.243,224.306,-60.933,-177.448,6.743,148.494
C06899=1194.239,224.553,-60.958,-177.445,6.746,148.494
C06900=1194.234,224.803,-60.983,-177.443,6.748,148.494
C06901=1194.230,225.052,-61.008,-177.440,6.749,148.493
C06902=1194.225,225.300,-61.034,-177.438,6.752,148.493
C06903=1194.221,225.549,-61.059,-177.435,6.754,148.493
C06904=1194.216,225.797,-61.084,-177.432,6.756,148.493
C06905=1194.212,226.046,-61.110,-177.430,6.758,148.493
C06906=1194.206,226.295,-61.135,-177.427,6.760,148.492
C06907=1194.202,226.544,-61.160,-177.424,6.763,148.492
C06908=1194.198,226.792,-61.186,-177.422,6.765,148.492
C06909=1194.193,227.041,-61.211,-177.419,6.767,148.492
C06910=1194.189,227.290,-61.237,-177.417,6.769,148.491
C06911=1194.185,227.538,-61.261,-177.414,6.772,148.491
C06912=1194.180,227.786,-61.287,-177.411,6.773,148.491
C06913=1194.176,228.035,-61.313,-177.409,6.775,148.490
C06914=1194.171,228.284,-61.338,-177.406,6.777,148.490
C06915=1194.167,228.533,-61.363,-177.403,6.780,148.490
C06916=1194.163,228.782,-61.389,-177.401,6.782,148.490
C06917=1194.158,229.030,-61.414,-177.398,6.784,148.490
C06918=1194.153,229.279,-61.440,-177.396,6.786,148.489
C06919=1194.149,229.527,-61.466,-177.393,6.788,148.489
C06920=1194.144,229.776,-61.491,-177.390,6.791,148.489
C06921=1194.140,230.025,-61.516,-177.388,6.792,148.489
C06922=1194.134,230.273,-61.542,-177.386,6.795,148.488
C06923=1194.130,230.522,-61.568,-177.382,6.797,148.488
C06924=1194.126,230.771,-61.594,-177.380,6.799,148.488
C06925=1194.121,231.019,-61.619,-177.378,6.801,148.488
C06926=1194.117,231.268,-61.645,-177.374,6.804,148.487
C06927=1194.113,231.517,-61.671,-177.372,6.806,148.487
C06928=1194.108,231.765,-61.696,-177.370,6.808,148.487
C06929=1194.104,232.014,-61.722,-177.367,6.810,148.487
C06930=1194.099,232.262,-61.748,-177.364,6.813,148.487
C06931=1194.095,232.511,-61.773,-177.361,6.815,148.486
C06932=1194.090,232.759,-61.799,-177.359,6.816,148.486
C06933=1194.085,233.008,-61.825,-177.356,6.819,148.486
C06934=1194.081,233.257,-61.851,-177.353,6.821,148.486
C06935=1194.076,233.505,-61.876,-177.351,6.823,148.486
C06936=1194.072,233.754,-61.902,-177.349,6.825,148.485
C06937=1194.068,234.003,-61.928,-177.346,6.828,148.485
C06938=1194.064,234.252,-61.953,-177.343,6.830,148.485
C06939=1194.059,234.500,-61.979,-177.341,6.832,148.484
C06940=1194.054,234.749,-62.005,-177.338,6.835,148.484
C06941=1194.050,234.998,-62.031,-177.335,6.837,148.484
C06942=1194.045,235.247,-62.057,-177.333,6.839,148.484
C06943=1194.041,235.494,-62.083,-177.330,6.841,148.484
C06944=1194.037,235.743,-62.109,-177.327,6.843,148.483
C06945=1194.032,235.992,-62.135,-177.325,6.845,148.483
C06946=1194.027,236.241,-62.161,-177.322,6.847,148.483
C06947=1194.022,236.511,-62.189,-177.320,6.850,148.483
C06948=1194.018,236.783,-62.217,-177.317,6.853,148.483
C06949=1194.013,237.055,-62.245,-177.314,6.855,148.482
C06950=1194.008,237.327,-62.274,-177.311,6.858,148.482
C06951=1194.003,237.575,-62.300,-177.309,6.860,148.482
C06952=1193.999,237.824,-62.326,-177.306,6.861,148.482
C06953=1193.994,238.072,-62.353,-177.303,6.864,148.482
C06954=1193.990,238.321,-62.378,-177.301,6.866,148.481
C06955=1193.986,238.570,-62.404,-177.298,6.868,148.481
C06956=1193.982,238.819,-62.430,-177.295,6.871,148.481
C06957=1193.976,239.066,-62.457,-177.293,6.873,148.481
C06958=1193.972,239.315,-62.482,-177.290,6.875,148.480
C06959=1193.968,239.564,-62.508,-177.288,6.878,148.480
C06960=1193.963,239.812,-62.535,-177.285,6.880,148.480
C06961=1193.959,240.061,-62.561,-177.283,6.882,148.480
C06962=1193.955,240.310,-62.587,-177.280,6.885,148.480
C06963=1193.949,240.558,-62.613,-177.278,6.887,148.480
C06964=1193.945,240.807,-62.639,-177.275,6.889,148.479
C06965=1193.941,241.055,-62.666,-177.272,6.891,148.479
C06966=1193.936,241.304,-62.692,-177.270,6.893,148.479
C06967=1193.932,241.553,-62.718,-177.267,6.895,148.478
C06968=1193.928,241.801,-62.745,-177.264,6.898,148.478
C06969=1193.923,242.050,-62.771,-177.262,6.900,148.478
C06970=1193.919,242.299,-62.798,-177.259,6.902,148.478
C06971=1193.914,242.547,-62.823,-177.256,6.905,148.478
C06972=1193.910,242.795,-62.849,-177.254,6.907,148.478
C06973=1193.905,243.044,-62.876,-177.251,6.909,148.477
C06974=1193.901,243.292,-62.902,-177.249,6.912,148.477
C06975=1193.896,243.541,-62.929,-177.246,6.914,148.477
C06976=1193.892,243.789,-62.955,-177.243,6.917,148.477
C06977=1193.887,244.039,-62.981,-177.241,6.919,148.477
C06978=1193.883,244.287,-63.008,-177.238,6.921,148.476
C06979=1193.878,244.536,-63.034,-177.235,6.923,148.476
C06980=1193.874,244.784,-63.061,-177.233,6.926,148.476
C06981=1193.870,245.032,-63.088,-177.230,6.927,148.476
C06982=1193.865,245.281,-63.113,-177.228,6.930,148.476
C06983=1193.861,245.530,-63.141,-177.226,6.933,148.476
C06984=1193.857,245.779,-63.166,-177.223,6.934,148.475
C06985=1193.852,246.027,-63.193,-177.220,6.937,148.475
C06986=1193.848,246.275,-63.220,-177.218,6.939,148.475
C06987=1193.843,246.524,-63.246,-177.215,6.942,148.475
C06988=1193.839,246.773,-63.273,-177.212,6.944,148.475
C06989=1193.834,247.021,-63.300,-177.210,6.946,148.474
C06990=1193.830,247.270,-63.326,-177.207,6.949,148.474
C06991=1193.826,247.518,-63.353,-177.205,6.951,148.474
C06992=1193.821,247.767,-63.380,-177.202,6.953,148.474
C06993=1193.817,248.015,-63.406,-177.199,6.956,148.474
C06994=1193.812,248.264,-63.432,-177.197,6.958,148.473
C06995=1193.807,248.513,-63.459,-177.194,6.961,148.473
C06996=1193.803,248.761,-63.486,-177.192,6.963,148.473
C06997=1193.799,249.009,-63.513,-177.189,6.965,148.473
C06998=1193.794,249.258,-63.540,-177.186,6.968,148.473
C06999=1193.790,249.507,-63.566,-177.184,6.970,148.473
C07000=1193.785,249.755,-63.593,-177.181,6.973,148.473
C07001=1193.781,250.003,-63.619,-177.179,6.974,148.472
C07002=1193.777,250.252,-63.646,-177.176,6.977,148.472
C07003=1193.772,250.500,-63.673,-177.173,6.979,148.472
C07004=1193.767,250.749,-63.701,-177.171,6.981,148.472
C07005=1193.763,250.998,-63.726,-177.168,6.984,148.472
C07006=1193.759,251.246,-63.753,-177.166,6.986,148.471
C07007=1193.754,251.495,-63.780,-177.163,6.988,148.471
C07008=1193.750,251.743,-63.807,-177.160,6.991,148.471
C07009=1193.745,251.991,-63.834,-177.158,6.993,148.471
C07010=1193.741,252.240,-63.861,-177.155,6.996,148.471
C07011=1193.736,252.488,-63.888,-177.153,6.998,148.471
C07012=1193.733,252.737,-63.915,-177.150,7.001,148.470
C07013=1193.728,252.986,-63.942,-177.147,7.003,148.470
C07014=1193.723,253.234,-63.969,-177.145,7.005,148.470
C07015=1193.719,253.483,-63.996,-177.143,7.008,148.470
C07016=1193.715,253.731,-64.023,-177.140,7.010,148.470
C07017=1193.710,253.979,-64.050,-177.137,7.013,148.470
C07018=1193.705,254.228,-64.077,-177.135,7.015,148.469
C07019=1193.701,254.476,-64.104,-177.132,7.018,148.469
C07020=1193.696,254.725,-64.131,-177.130,7.020,148.469
C07021=1193.693,254.974,-64.158,-177.127,7.022,148.469
C07022=1193.688,255.222,-64.185,-177.124,7.025,148.469
C07023=1193.684,255.471,-64.212,-177.122,7.027,148.469
C07024=1193.679,255.719,-64.239,-177.119,7.029,148.468
C07025=1193.674,255.967,-64.267,-177.117,7.032,148.468
C07026=1193.670,256.216,-64.294,-177.114,7.034,148.468
C07027=1193.667,256.464,-64.320,-177.111,7.036,148.468
C07028=1193.662,256.713,-64.348,-177.109,7.039,148.468
C07029=1193.657,256.961,-64.375,-177.106,7.041,148.468
C07030=1193.653,257.210,-64.402,-177.104,7.043,148.468
C07031=1193.648,257.458,-64.429,-177.101,7.046,148.467
C07032=1193.644,257.706,-64.456,-177.099,7.048,148.467
C07033=1193.639,257.956,-64.484,-177.096,7.051,148.467
C07034=1193.635,258.204,-64.511,-177.093,7.053,148.467
C07035=1193.630,258.452,-64.538,-177.091,7.056,148.467
C07036=1193.626,258.700,-64.566,-177.088,7.058,148.467
C07037=1193.621,258.949,-64.593,-177.085,7.061,148.466
C07038=1193.617,259.198,-64.620,-177.083,7.063,148.466
C07039=1193.612,259.447,-64.647,-177.080,7.066,148.466
C07040=1193.609,259.694,-64.675,-177.078,7.068,148.466
C07041=1193.604,259.943,-64.702,-177.075,7.071,148.466
C07042=1193.600,260.192,-64.729,-177.073,7.073,148.466
C07043=1193.596,260.440,-64.757,-177.070,7.075,148.466
C07044=1193.591,260.688,-64.784,-177.067,7.078,148.466
C07045=1193.586,260.937,-64.811,-177.065,7.080,148.465
C07046=1193.583,261.185,-64.839,-177.062,7.083,148.465
C07047=1193.578,261.434,-64.866,-177.060,7.085,148.465
C07048=1193.573,261.682,-64.894,-177.057,7.088,148.465
C07049=1193.568,261.930,-64.922,-177.055,7.090,148.465
C07050=1193.564,262.180,-64.949,-177.052,7.093,148.465
C07051=1193.560,262.452,-64.979,-177.049,7.096,148.465
C07052=1193.555,262.725,-65.009,-177.047,7.098,148.464
C07053=1193.550,262.998,-65.040,-177.044,7.101,148.464
C07054=1193.545,263.270,-65.069,-177.041,7.103,148.464
C07055=1193.541,263.519,-65.098,-177.038,7.106,148.464
C07056=1193.536,263.768,-65.125,-177.036,7.109,148.464
C07057=1193.532,264.015,-65.153,-177.033,7.111,148.464
C07058=1193.528,264.265,-65.180,-177.030,7.113,148.464
C07059=1193.523,264.513,-65.208,-177.028,7.116,148.464
C07060=1193.519,264.761,-65.235,-177.025,7.118,148.463
C07061=1193.515,265.010,-65.263,-177.022,7.121,148.463
C07062=1193.510,265.258,-65.290,-177.020,7.123,148.463
C07063=1193.505,265.506,-65.319,-177.018,7.126,148.463
C07064=1193.501,265.755,-65.347,-177.015,7.128,148.463
C07065=1193.497,266.003,-65.374,-177.012,7.131,148.463
C07066=1193.492,266.251,-65.402,-177.010,7.133,148.463
C07067=1193.489,266.500,-65.430,-177.007,7.136,148.462
C07068=1193.483,266.749,-65.458,-177.005,7.138,148.462
C07069=1193.479,266.996,-65.485,-177.002,7.141,148.462
C07070=1193.475,267.246,-65.513,-177.000,7.143,148.462
C07071=1193.471,267.494,-65.541,-176.997,7.146,148.462
C07072=1193.467,267.742,-65.569,-176.994,7.148,148.462
C07073=1193.462,267.990,-65.597,-176.992,7.151,148.462
C07074=1193.457,268.239,-65.624,-176.990,7.153,148.462
C07075=1193.453,268.487,-65.652,-176.986,7.156,148.461
C07076=1193.449,268.735,-65.680,-176.984,7.159,148.461
C07077=1193.444,268.984,-65.709,-176.982,7.161,148.461
C07078=1193.440,269.233,-65.736,-176.979,7.164,148.461
C07079=1193.435,269.481,-65.764,-176.976,7.166,148.461
C07080=1193.431,269.729,-65.792,-176.974,7.169,148.461
C07081=1193.427,269.977,-65.820,-176.971,7.171,148.461
C07082=1193.423,270.226,-65.848,-176.969,7.174,148.461
C07083=1193.418,270.474,-65.875,-176.966,7.176,148.460
C07084=1193.414,270.723,-65.904,-176.963,7.179,148.460
C07085=1193.409,270.971,-65.932,-176.961,7.181,148.460
C07086=1193.404,271.219,-65.960,-176.958,7.184,148.460
C07087=1193.401,271.468,-65.988,-176.956,7.186,148.460
C07088=1193.396,271.716,-66.016,-176.953,7.189,148.460
C07089=1193.392,271.965,-66.045,-176.950,7.192,148.460
C07090=1193.387,272.213,-66.073,-176.948,7.194,148.460
C07091=1193.383,272.462,-66.100,-176.945,7.197,148.460
C07092=1193.378,272.710,-66.129,-176.943,7.199,148.460
C07093=1193.374,272.959,-66.157,-176.940,7.202,148.459
C07094=1193.369,273.207,-66.185,-176.938,7.204,148.459
C07095=1193.366,273.455,-66.213,-176.935,7.207,148.459
C07096=1193.361,273.703,-66.241,-176.932,7.210,148.459
C07097=1193.357,273.952,-66.270,-176.930,7.212,148.459
C07098=1193.352,274.200,-66.297,-176.927,7.215,148.459
C07099=1193.348,274.449,-66.326,-176.925,7.217,148.459
C07100=1193.344,274.697,-66.354,-176.922,7.220,148.459
C07101=1193.339,274.946,-66.383,-176.920,7.222,148.459
C07102=1193.335,275.193,-66.410,-176.917,7.225,148.459
C07103=1193.331,275.442,-66.440,-176.914,7.228,148.458
C07104=1193.327,275.690,-66.468,-176.912,7.230,148.458
C07105=1193.322,275.938,-66.496,-176.909,7.233,148.458
C07106=1193.318,276.187,-66.525,-176.907,7.235,148.458
C07107=1193.313,276.435,-66.553,-176.904,7.238,148.458
C07108=1193.309,276.684,-66.581,-176.902,7.240,148.458
C07109=1193.304,276.932,-66.609,-176.899,7.243,148.458
C07110=1193.300,277.181,-66.638,-176.897,7.246,148.458
C07111=1193.296,277.429,-66.667,-176.894,7.249,148.458
C07112=1193.292,277.677,-66.695,-176.891,7.251,148.458
C07113=1193.287,277.926,-66.724,-176.889,7.253,148.457
C07114=1193.283,278.173,-66.751,-176.886,7.256,148.457
C07115=1193.279,278.422,-66.781,-176.884,7.259,148.457
C07116=1193.275,278.670,-66.809,-176.882,7.262,148.457
C07117=1193.270,278.918,-66.837,-176.879,7.265,148.457
C07118=1193.265,279.167,-66.866,-176.876,7.266,148.457
C07119=1193.261,279.415,-66.895,-176.873,7.269,148.457
C07120=1193.257,279.664,-66.923,-176.871,7.272,148.457
C07121=1193.253,279.912,-66.951,-176.869,7.275,148.457
C07122=1193.248,280.160,-66.980,-176.866,7.278,148.457
C07123=1193.244,280.409,-67.009,-176.864,7.280,148.457
C07124=1193.240,280.657,-67.037,-176.861,7.283,148.457
C07125=1193.235,280.905,-67.066,-176.858,7.286,148.456
C07126=1193.231,281.154,-67.095,-176.856,7.288,148.456
C07127=1193.227,281.402,-67.123,-176.853,7.291,148.456
C07128=1193.222,281.650,-67.152,-176.850,7.294,148.456
C07129=1193.218,281.899,-67.181,-176.848,7.296,148.456
C07130=1193.214,282.147,-67.209,-176.845,7.299,148.456
C07131=1193.209,282.395,-67.238,-176.843,7.301,148.456
C07132=1193.205,282.644,-67.267,-176.841,7.304,148.456
C07133=1193.201,282.892,-67.297,-176.837,7.307,148.456
C07134=1193.196,283.140,-67.324,-176.835,7.309,148.456
C07135=1193.192,283.388,-67.354,-176.833,7.312,148.456
C07136=1193.188,283.637,-67.383,-176.830,7.315,148.456
C07137=1193.183,283.885,-67.412,-176.828,7.317,148.456
C07138=1193.179,284.133,-67.440,-176.825,7.320,148.456
C07139=1193.175,284.381,-67.469,-176.823,7.322,148.456
C07140=1193.170,284.630,-67.498,-176.820,7.325,148.456
C07141=1193.166,284.878,-67.527,-176.817,7.328,148.455
C07142=1193.162,285.126,-67.555,-176.815,7.330,148.455
C07143=1193.158,285.375,-67.585,-176.812,7.333,148.455
C07144=1193.153,285.622,-67.614,-176.809,7.336,148.455
C07145=1193.148,285.871,-67.643,-176.807,7.338,148.455
C07146=1193.144,286.119,-67.672,-176.805,7.341,148.455
C07147=1193.140,286.368,-67.701,-176.802,7.344,148.455
C07148=1193.136,286.616,-67.729,-176.800,7.347,148.455
C07149=1193.132,286.864,-67.759,-176.797,7.350,148.455
C07150=1193.127,287.113,-67.787,-176.795,7.352,148.455
C07151=1193.123,287.361,-67.817,-176.792,7.355,148.455
C07152=1193.119,287.609,-67.846,-176.789,7.358,148.455
C07153=1193.114,287.857,-67.875,-176.787,7.360,148.455
C07154=1193.109,288.106,-67.904,-176.785,7.363,148.455
C07155=1193.105,288.380,-67.936,-176.781,7.366,148.454
C07156=1193.101,288.654,-67.968,-176.779,7.369,148.454
C07157=1193.095,288.929,-68.001,-176.776,7.372,148.454
C07158=1193.091,289.203,-68.033,-176.773,7.375,148.454
C07159=1193.086,289.452,-68.062,-176.771,7.378,148.454
C07160=1193.082,289.700,-68.091,-176.768,7.381,148.454
C07161=1193.078,289.948,-68.121,-176.766,7.383,148.454
C07162=1193.074,290.197,-68.150,-176.763,7.386,148.454
C07163=1193.069,290.445,-68.180,-176.760,7.389,148.454
C07164=1193.064,290.693,-68.208,-176.758,7.391,148.454
C07165=1193.060,290.941,-68.237,-176.755,7.394,148.454
C07166=1193.056,291.190,-68.267,-176.753,7.397,148.454
C07167=1193.052,291.438,-68.296,-176.751,7.399,148.454
C07168=1193.048,291.686,-68.326,-176.748,7.402,148.454
C07169=1193.043,291.934,-68.355,-176.745,7.405,148.454
C07170=1193.039,292.183,-68.385,-176.743,7.407,148.454
C07171=1193.035,292.430,-68.414,-176.740,7.410,148.454
C07172=1193.030,292.678,-68.443,-176.738,7.413,148.454
C07173=1193.026,292.927,-68.473,-176.735,7.416,148.454
C07174=1193.022,293.175,-68.502,-176.733,7.419,148.454
C07175=1193.018,293.423,-68.532,-176.730,7.422,148.454
C07176=1193.014,293.672,-68.561,-176.728,7.424,148.454
C07177=1193.009,293.920,-68.591,-176.725,7.427,148.454
C07178=1193.005,294.168,-68.620,-176.722,7.430,148.454
C07179=1193.001,294.416,-68.649,-176.720,7.433,148.454
C07180=1192.997,294.665,-68.679,-176.718,7.435,148.453
C07181=1192.992,294.913,-68.709,-176.715,7.438,148.453
C07182=1192.987,295.161,-68.738,-176.712,7.441,148.453
C07183=1192.983,295.409,-68.767,-176.710,7.443,148.453
C07184=1192.979,295.657,-68.797,-176.707,7.446,148.453
C07185=1192.975,295.906,-68.826,-176.705,7.449,148.453
C07186=1192.970,296.154,-68.856,-176.702,7.451,148.453
C07187=1192.966,296.402,-68.885,-176.700,7.454,148.453
C07188=1192.962,296.650,-68.916,-176.697,7.457,148.453
C07189=1192.957,296.898,-68.946,-176.694,7.460,148.453
C07190=1192.953,297.147,-68.975,-176.692,7.463,148.453
C07191=1192.949,297.395,-69.004,-176.689,7.466,148.453
C07192=1192.945,297.643,-69.034,-176.687,7.469,148.453
C07193=1192.940,297.891,-69.065,-176.685,7.471,148.453
C07194=1192.936,298.139,-69.094,-176.682,7.474,148.453
C07195=1192.932,298.388,-69.124,-176.679,7.477,148.453
C07196=1192.928,298.636,-69.153,-176.677,7.480,148.453
C07197=1192.924,298.884,-69.182,-176.674,7.482,148.453
C07198=1192.919,299.132,-69.213,-176.672,7.485,148.453
C07199=1192.915,299.380,-69.243,-176.669,7.488,148.453
C07200=1192.911,299.629,-69.272,-176.667,7.490,148.453
C07201=1192.906,299.877,-69.303,-176.664,7.493,148.453
C07202=1192.902,300.125,-69.332,-176.662,7.496,148.453
C07203=1192.898,300.373,-69.362,-176.659,7.499,148.453
C07204=1192.894,300.621,-69.392,-176.657,7.502,148.453
C07205=1192.889,300.869,-69.422,-176.654,7.505,148.453
C07206=1192.885,301.118,-69.451,-176.652,7.508,148.453
C07207=1192.881,301.365,-69.482,-176.649,7.510,148.453
C07208=1192.876,301.614,-69.512,-176.647,7.513,148.453
C07209=1192.872,301.861,-69.542,-176.644,7.516,148.453
C07210=1192.868,302.110,-69.572,-176.641,7.519,148.453
C07211=1192.864,302.358,-69.602,-176.639,7.521,148.453
C07212=1192.860,302.607,-69.632,-176.637,7.524,148.453
C07213=1192.855,302.855,-69.662,-176.634,7.527,148.453
C07214=1192.851,303.103,-69.692,-176.632,7.530,148.453
C07215=1192.847,303.351,-69.722,-176.629,7.533,148.453
C07216=1192.842,303.599,-69.752,-176.627,7.536,148.453
C07217=1192.838,303.847,-69.782,-176.624,7.539,148.453
C07218=1192.833,304.095,-69.813,-176.621,7.542,148.453
C07219=1192.829,304.344,-69.842,-176.619,7.544,148.453
C07220=1192.825,304.591,-69.872,-176.616,7.547,148.453
C07221=1192.821,304.840,-69.903,-176.614,7.550,148.453
C07222=1192.817,305.088,-69.933,-176.612,7.552,148.453
C07223=1192.812,305.336,-69.964,-176.609,7.555,148.453
C07224=1192.808,305.584,-69.993,-176.607,7.558,148.453
C07225=1192.804,305.832,-70.024,-176.604,7.561,148.453
C07226=1192.800,306.080,-70.054,-176.602,7.563,148.453
C07227=1192.795,306.329,-70.084,-176.600,7.567,148.453
C07228=1192.792,306.577,-70.114,-176.597,7.570,148.453
C07229=1192.787,306.825,-70.145,-176.594,7.573,148.453
C07230=1192.783,307.073,-70.175,-176.592,7.575,148.453
C07231=1192.778,307.321,-70.205,-176.589,7.578,148.453
C07232=1192.774,307.569,-70.236,-176.587,7.581,148.453
C07233=1192.769,307.817,-70.266,-176.584,7.584,148.453
C07234=1192.765,308.066,-70.297,-176.582,7.587,148.453
C07235=1192.761,308.314,-70.327,-176.580,7.590,148.453
C07236=1192.757,308.562,-70.358,-176.577,7.593,148.453
C07237=1192.753,308.810,-70.387,-176.574,7.596,148.453
C07238=1192.748,309.058,-70.418,-176.572,7.599,148.453
C07239=1192.745,309.306,-70.448,-176.570,7.601,148.453
C07240=1192.740,309.554,-70.479,-176.567,7.604,148.453
C07241=1192.736,309.802,-70.510,-176.564,7.607,148.453
C07242=1192.731,310.050,-70.539,-176.562,7.610,148.453
C07243=1192.727,310.298,-70.570,-176.560,7.613,148.453
C07244=1192.723,310.547,-70.601,-176.557,7.616,148.453
C07245=1192.719,310.795,-70.632,-176.555,7.619,148.453
C07246=1192.714,311.043,-70.662,-176.552,7.622,148.453
C07247=1192.710,311.290,-70.692,-176.550,7.624,148.453
C07248=1192.706,311.539,-70.724,-176.547,7.627,148.453
C07249=1192.702,311.787,-70.754,-176.545,7.630,148.453
C07250=1192.698,312.035,-70.785,-176.542,7.633,148.453
C07251=1192.693,312.283,-70.815,-176.539,7.636,148.453
C07252=1192.689,312.532,-70.846,-176.538,7.639,148.453
C07253=1192.684,312.780,-70.876,-176.535,7.642,148.453
C07254=1192.680,313.027,-70.907,-176.532,7.645,148.453
C07255=1192.676,313.276,-70.938,-176.530,7.648,148.453
C07256=1192.672,313.524,-70.969,-176.528,7.650,148.453
C07257=1192.668,313.772,-70.999,-176.525,7.653,148.453
C07258=1192.663,314.020,-71.029,-176.522,7.656,148.453
C07259=1192.659,314.296,-71.064,-176.520,7.659,148.453
C07260=1192.654,314.572,-71.098,-176.518,7.663,148.454
C07261=1192.649,314.849,-71.133,-176.514,7.666,148.454
C07262=1192.644,315.125,-71.167,-176.512,7.669,148.454
C07263=1192.640,315.374,-71.198,-176.509,7.672,148.454
C07264=1192.636,315.621,-71.228,-176.507,7.675,148.454
C07265=1192.632,315.869,-71.259,-176.505,7.678,148.454
C07266=1192.628,316.117,-71.291,-176.502,7.681,148.454
C07267=1192.624,316.365,-71.322,-176.500,7.684,148.454
C07268=1192.619,316.613,-71.353,-176.497,7.687,148.454
C07269=1192.616,316.862,-71.383,-176.495,7.689,148.454
C07270=1192.611,317.110,-71.414,-176.492,7.693,148.454
C07271=1192.607,317.358,-71.446,-176.490,7.696,148.454
C07272=1192.603,317.606,-71.477,-176.487,7.699,148.454
C07273=1192.598,317.854,-71.507,-176.485,7.701,148.454
C07274=1192.594,318.102,-71.538,-176.483,7.704,148.454
C07275=1192.589,318.350,-71.569,-176.480,7.707,148.454
C07276=1192.586,318.598,-71.601,-176.478,7.711,148.454
C07277=1192.582,318.846,-71.631,-176.475,7.714,148.454
C07278=1192.577,319.094,-71.662,-176.473,7.716,148.454
C07279=1192.574,319.342,-71.694,-176.471,7.719,148.455
C07280=1192.569,319.590,-71.725,-176.468,7.722,148.455
C07281=1192.565,319.839,-71.756,-176.465,7.725,148.455
C07282=1192.561,320.086,-71.787,-176.463,7.729,148.455
C07283=1192.556,320.334,-71.818,-176.461,7.731,148.455
C07284=1192.552,320.582,-71.849,-176.459,7.734,148.455
C07285=1192.548,320.830,-71.881,-176.456,7.737,148.455
C07286=1192.544,321.078,-71.912,-176.453,7.740,148.455
C07287=1192.539,321.326,-71.943,-176.451,7.743,148.455
C07288=1192.535,321.574,-71.974,-176.449,7.746,148.455
C07289=1192.531,321.822,-72.006,-176.447,7.749,148.455
C07290=1192.527,322.070,-72.037,-176.444,7.752,148.455
C07291=1192.522,322.318,-72.068,-176.441,7.755,148.455
C07292=1192.519,322.566,-72.100,-176.439,7.758,148.456
C07293=1192.514,322.814,-72.130,-176.437,7.760,148.455
C07294=1192.510,323.062,-72.162,-176.435,7.764,148.456
C07295=1192.506,323.310,-72.193,-176.432,7.767,148.456
C07296=1192.502,323.558,-72.225,-176.430,7.770,148.456
C07297=1192.498,323.806,-72.256,-176.427,7.773,148.456
C07298=1192.494,324.054,-72.287,-176.425,7.775,148.456
C07299=1192.489,324.302,-72.319,-176.423,7.779,148.456
C07300=1192.485,324.550,-72.350,-176.420,7.782,148.456
C07301=1192.481,324.798,-72.381,-176.418,7.785,148.456
C07302=1192.477,325.046,-72.413,-176.415,7.788,148.456
C07303=1192.473,325.294,-72.444,-176.413,7.791,148.456
C07304=1192.468,325.542,-72.476,-176.411,7.794,148.456
C07305=1192.464,325.790,-72.507,-176.408,7.797,148.457
C07306=1192.460,326.038,-72.539,-176.406,7.800,148.457
C07307=1192.456,326.285,-72.571,-176.403,7.803,148.457
C07308=1192.452,326.534,-72.602,-176.401,7.806,148.457
C07309=1192.447,326.781,-72.633,-176.399,7.809,148.457
C07310=1192.444,327.029,-72.665,-176.396,7.812,148.457
C07311=1192.439,327.278,-72.697,-176.394,7.815,148.457
C07312=1192.435,327.526,-72.728,-176.391,7.818,148.457
C07313=1192.431,327.774,-72.760,-176.389,7.821,148.457
C07314=1192.427,328.021,-72.792,-176.386,7.824,148.457
C07315=1192.423,328.270,-72.823,-176.385,7.827,148.458
C07316=1192.418,328.517,-72.855,-176.382,7.830,148.458
C07317=1192.414,328.766,-72.887,-176.380,7.833,148.458
C07318=1192.410,329.014,-72.918,-176.377,7.836,148.458
C07319=1192.406,329.261,-72.950,-176.375,7.840,148.458
C07320=1192.401,329.510,-72.982,-176.373,7.842,148.458
